	VAR robtarget OpenholeUD_5476 := [[469.92, -36.3, 185.04], [0.127117, 0.695587, 0.707021, -0.011034], [0,0,0,0], [9E9, 9E9, 9E9, 9E9, 9E9, 9E9]];
	VAR robtarget OpenholeUD_5477 := [[465.97, -36.3, 184.38], [0.114661, 0.697748, 0.707103, 0.002317], [0,0,0,0], [9E9, 9E9, 9E9, 9E9, 9E9, 9E9]];
	VAR robtarget OpenholeUD_5478 := [[462.03, -36.3, 183.73], [0.101936, 0.699721, 0.706932, 0.015742], [0,0,0,0], [9E9, 9E9, 9E9, 9E9, 9E9, 9E9]];
	VAR robtarget OpenholeUD_5479 := [[458.08, -36.3, 183.07], [0.088974, 0.701487, 0.706504, 0.029202], [0,0,0,0], [9E9, 9E9, 9E9, 9E9, 9E9, 9E9]];
	VAR robtarget OpenholeUD_5480 := [[454.14, -36.3, 182.42], [0.075811, 0.703031, 0.705819, 0.042651], [0,0,0,0], [9E9, 9E9, 9E9, 9E9, 9E9, 9E9]];
	VAR robtarget OpenholeUD_5481 := [[450.19, -36.3, 181.76], [0.062487, 0.70434, 0.704882, 0.056046], [0,0,0,0], [9E9, 9E9, 9E9, 9E9, 9E9, 9E9]];
	VAR robtarget OpenholeUD_5482 := [[446.24, -36.3, 181.11], [0.049045, 0.705404, 0.703698, 0.069344], [0,0,0,0], [9E9, 9E9, 9E9, 9E9, 9E9, 9E9]];
	VAR robtarget OpenholeUD_5483 := [[442.3, -36.3, 180.45], [0.035527, 0.706214, 0.702277, 0.082504], [0,0,0,0], [9E9, 9E9, 9E9, 9E9, 9E9, 9E9]];
	VAR robtarget OpenholeUD_5484 := [[438.35, -36.3, 179.79], [0.021978, 0.706765, 0.70063, 0.095485], [0,0,0,0], [9E9, 9E9, 9E9, 9E9, 9E9, 9E9]];
	VAR robtarget OpenholeUD_5485 := [[434.41, -36.3, 179.14], [0.008444, 0.707056, 0.698772, 0.10825], [0,0,0,0], [9E9, 9E9, 9E9, 9E9, 9E9, 9E9]];
	VAR robtarget OpenholeUD_5486 := [[430.46, -36.3, 178.48], [-0.005032, 0.707089, 0.696718, 0.120767], [0,0,0,0], [9E9, 9E9, 9E9, 9E9, 9E9, 9E9]];
	VAR robtarget OpenholeUD_5487 := [[426.52, -36.3, 177.83], [-0.018407, 0.706867, 0.694485, 0.133005], [0,0,0,0], [9E9, 9E9, 9E9, 9E9, 9E9, 9E9]];
	VAR robtarget OpenholeUD_5488 := [[422.57, -36.3, 177.17], [-0.03164, 0.706399, 0.692093, 0.144938], [0,0,0,0], [9E9, 9E9, 9E9, 9E9, 9E9, 9E9]];
	VAR robtarget OpenholeUD_5489 := [[418.62, -36.3, 176.52], [-0.044695, 0.705693, 0.68956, 0.156545], [0,0,0,0], [9E9, 9E9, 9E9, 9E9, 9E9, 9E9]];
	VAR robtarget OpenholeUD_5490 := [[414.68, -36.3, 175.86], [-0.057536, 0.704762, 0.686906, 0.167808], [0,0,0,0], [9E9, 9E9, 9E9, 9E9, 9E9, 9E9]];
	VAR robtarget OpenholeUD_5491 := [[410.73, -36.3, 175.2], [-0.070134, 0.70362, 0.68415, 0.178714], [0,0,0,0], [9E9, 9E9, 9E9, 9E9, 9E9, 9E9]];
	VAR robtarget OpenholeUD_5492 := [[406.79, -36.3, 174.55], [-0.082462, 0.702282, 0.68131, 0.189254], [0,0,0,0], [9E9, 9E9, 9E9, 9E9, 9E9, 9E9]];
	VAR robtarget OpenholeUD_5493 := [[402.84, -36.3, 173.89], [-0.094498, 0.700764, 0.678404, 0.199421], [0,0,0,0], [9E9, 9E9, 9E9, 9E9, 9E9, 9E9]];
	VAR robtarget OpenholeUD_5494 := [[398.89, -36.3, 173.24], [-0.106223, 0.699083, 0.675448, 0.209213], [0,0,0,0], [9E9, 9E9, 9E9, 9E9, 9E9, 9E9]];
	VAR robtarget OpenholeUD_5495 := [[394.95, -36.3, 172.58], [-0.117622, 0.697255, 0.672458, 0.218631], [0,0,0,0], [9E9, 9E9, 9E9, 9E9, 9E9, 9E9]];
	VAR robtarget OpenholeUD_5496 := [[389.32, -36.3, 171.65], [-0.13331, 0.694427, 0.66816, 0.231434], [0,0,0,0], [9E9, 9E9, 9E9, 9E9, 9E9, 9E9]];
	VAR robtarget OpenholeUD_5497 := [[385.32, -36.3, 171.66], [-0.183051, 0.683002, 0.683002, 0.183051], [0,0,0,0], [9E9, 9E9, 9E9, 9E9, 9E9, 9E9]];
	VAR robtarget OpenholeUD_5498 := [[381.32, -36.3, 171.67], [-0.183051, 0.683002, 0.683002, 0.183051], [0,0,0,0], [9E9, 9E9, 9E9, 9E9, 9E9, 9E9]];
	VAR robtarget OpenholeUD_5499 := [[377.32, -36.3, 171.68], [-0.183051, 0.683002, 0.683002, 0.183051], [0,0,0,0], [9E9, 9E9, 9E9, 9E9, 9E9, 9E9]];
	VAR robtarget OpenholeUD_5500 := [[373.32, -36.3, 171.7], [-0.183051, 0.683002, 0.683002, 0.183051], [0,0,0,0], [9E9, 9E9, 9E9, 9E9, 9E9, 9E9]];
	VAR robtarget OpenholeUD_5501 := [[369.32, -36.3, 171.71], [-0.183051, 0.683002, 0.683002, 0.183051], [0,0,0,0], [9E9, 9E9, 9E9, 9E9, 9E9, 9E9]];
	VAR robtarget OpenholeUD_5502 := [[369.32, -36.3, 171.71], [-0.183051, 0.683002, 0.683002, 0.183051], [0,0,0,0], [9E9, 9E9, 9E9, 9E9, 9E9, 9E9]];
	VAR robtarget OpenholeUD_5503 := [[369.31, -37.5, 171.02], [-0.183051, 0.683002, 0.683002, 0.183051], [0,0,0,0], [9E9, 9E9, 9E9, 9E9, 9E9, 9E9]];
	VAR robtarget OpenholeUD_5504 := [[373.31, -37.5, 171], [-0.183051, 0.683002, 0.683002, 0.183051], [0,0,0,0], [9E9, 9E9, 9E9, 9E9, 9E9, 9E9]];
	VAR robtarget OpenholeUD_5505 := [[377.31, -37.5, 170.99], [-0.183051, 0.683002, 0.683002, 0.183051], [0,0,0,0], [9E9, 9E9, 9E9, 9E9, 9E9, 9E9]];
	VAR robtarget OpenholeUD_5506 := [[381.31, -37.5, 170.98], [-0.183051, 0.683002, 0.683002, 0.183051], [0,0,0,0], [9E9, 9E9, 9E9, 9E9, 9E9, 9E9]];
	VAR robtarget OpenholeUD_5507 := [[385.31, -37.5, 170.97], [-0.183051, 0.683002, 0.683002, 0.183051], [0,0,0,0], [9E9, 9E9, 9E9, 9E9, 9E9, 9E9]];
	VAR robtarget OpenholeUD_5508 := [[389.31, -37.5, 170.95], [-0.129902, 0.695072, 0.667021, 0.234697], [0,0,0,0], [9E9, 9E9, 9E9, 9E9, 9E9, 9E9]];
	VAR robtarget OpenholeUD_5509 := [[393.25, -37.5, 171.65], [-0.118943, 0.697031, 0.670055, 0.225889], [0,0,0,0], [9E9, 9E9, 9E9, 9E9, 9E9, 9E9]];
	VAR robtarget OpenholeUD_5510 := [[397.19, -37.5, 172.35], [-0.107648, 0.698865, 0.673079, 0.216713], [0,0,0,0], [9E9, 9E9, 9E9, 9E9, 9E9, 9E9]];
	VAR robtarget OpenholeUD_5511 := [[401.13, -37.5, 173.05], [-0.096026, 0.700556, 0.676079, 0.207165], [0,0,0,0], [9E9, 9E9, 9E9, 9E9, 9E9, 9E9]];
	VAR robtarget OpenholeUD_5512 := [[405.07, -37.5, 173.75], [-0.084089, 0.702089, 0.679041, 0.197241], [0,0,0,0], [9E9, 9E9, 9E9, 9E9, 9E9, 9E9]];
	VAR robtarget OpenholeUD_5513 := [[409, -37.5, 174.45], [-0.071857, 0.703446, 0.681948, 0.186942], [0,0,0,0], [9E9, 9E9, 9E9, 9E9, 9E9, 9E9]];
	VAR robtarget OpenholeUD_5514 := [[412.94, -37.5, 175.15], [-0.059348, 0.704612, 0.684783, 0.176273], [0,0,0,0], [9E9, 9E9, 9E9, 9E9, 9E9, 9E9]];
	VAR robtarget OpenholeUD_5515 := [[416.88, -37.5, 175.85], [-0.04659, 0.70557, 0.687529, 0.165241], [0,0,0,0], [9E9, 9E9, 9E9, 9E9, 9E9, 9E9]];
	VAR robtarget OpenholeUD_5516 := [[420.82, -37.5, 176.55], [-0.03361, 0.706308, 0.690166, 0.153855], [0,0,0,0], [9E9, 9E9, 9E9, 9E9, 9E9, 9E9]];
	VAR robtarget OpenholeUD_5517 := [[424.76, -37.5, 177.25], [-0.020441, 0.706811, 0.692675, 0.142133], [0,0,0,0], [9E9, 9E9, 9E9, 9E9, 9E9, 9E9]];
	VAR robtarget OpenholeUD_5518 := [[428.7, -37.5, 177.95], [-0.00712, 0.707071, 0.695037, 0.130091], [0,0,0,0], [9E9, 9E9, 9E9, 9E9, 9E9, 9E9]];
	VAR robtarget OpenholeUD_5519 := [[432.63, -37.5, 178.65], [0.006313, 0.707079, 0.697233, 0.117755], [0,0,0,0], [9E9, 9E9, 9E9, 9E9, 9E9, 9E9]];
	VAR robtarget OpenholeUD_5520 := [[436.57, -37.5, 179.35], [0.019818, 0.706829, 0.699245, 0.105152], [0,0,0,0], [9E9, 9E9, 9E9, 9E9, 9E9, 9E9]];
	VAR robtarget OpenholeUD_5521 := [[440.51, -37.5, 180.05], [0.03335, 0.70632, 0.701055, 0.092312], [0,0,0,0], [9E9, 9E9, 9E9, 9E9, 9E9, 9E9]];
	VAR robtarget OpenholeUD_5522 := [[444.45, -37.5, 180.75], [0.046866, 0.705552, 0.702649, 0.079272], [0,0,0,0], [9E9, 9E9, 9E9, 9E9, 9E9, 9E9]];
	VAR robtarget OpenholeUD_5523 := [[448.39, -37.5, 181.45], [0.06032, 0.704529, 0.704013, 0.066068], [0,0,0,0], [9E9, 9E9, 9E9, 9E9, 9E9, 9E9]];
	VAR robtarget OpenholeUD_5524 := [[452.33, -37.5, 182.15], [0.073668, 0.703259, 0.705137, 0.052743], [0,0,0,0], [9E9, 9E9, 9E9, 9E9, 9E9, 9E9]];
	VAR robtarget OpenholeUD_5525 := [[456.26, -37.5, 182.85], [0.086868, 0.701751, 0.706012, 0.039337], [0,0,0,0], [9E9, 9E9, 9E9, 9E9, 9E9, 9E9]];
	VAR robtarget OpenholeUD_5526 := [[460.2, -37.5, 183.55], [0.09988, 0.700017, 0.706633, 0.025894], [0,0,0,0], [9E9, 9E9, 9E9, 9E9, 9E9, 9E9]];
	VAR robtarget OpenholeUD_5527 := [[464.14, -37.5, 184.25], [0.112666, 0.698073, 0.706997, 0.012458], [0,0,0,0], [9E9, 9E9, 9E9, 9E9, 9E9, 9E9]];
	VAR robtarget OpenholeUD_5528 := [[468.08, -37.5, 184.95], [0.125192, 0.695936, 0.707106, -0.000928], [0,0,0,0], [9E9, 9E9, 9E9, 9E9, 9E9, 9E9]];
	VAR robtarget OpenholeUD_5529 := [[472.02, -37.5, 185.65], [0.13743, 0.693623, 0.706964, -0.014223], [0,0,0,0], [9E9, 9E9, 9E9, 9E9, 9E9, 9E9]];
	VAR robtarget OpenholeUD_5530 := [[475.96, -37.5, 186.35], [0.149352, 0.691154, 0.706576, -0.027387], [0,0,0,0], [9E9, 9E9, 9E9, 9E9, 9E9, 9E9]];
	VAR robtarget OpenholeUD_5531 := [[479.89, -37.5, 187.05], [0.160938, 0.688548, 0.705953, -0.040383], [0,0,0,0], [9E9, 9E9, 9E9, 9E9, 9E9, 9E9]];
	VAR robtarget OpenholeUD_5532 := [[483.83, -37.5, 187.75], [0.172171, 0.685826, 0.705104, -0.053177], [0,0,0,0], [9E9, 9E9, 9E9, 9E9, 9E9, 9E9]];
	VAR robtarget OpenholeUD_5533 := [[487.77, -37.5, 188.45], [0.183038, 0.683006, 0.704044, -0.06574], [0,0,0,0], [9E9, 9E9, 9E9, 9E9, 9E9, 9E9]];
	VAR robtarget OpenholeUD_5534 := [[491.71, -37.5, 189.15], [0.193531, 0.680107, 0.702787, -0.078043], [0,0,0,0], [9E9, 9E9, 9E9, 9E9, 9E9, 9E9]];
	VAR robtarget OpenholeUD_5535 := [[495.65, -37.5, 189.85], [0.203644, 0.677148, 0.701347, -0.090066], [0,0,0,0], [9E9, 9E9, 9E9, 9E9, 9E9, 9E9]];
	VAR robtarget OpenholeUD_5536 := [[499.59, -37.5, 190.55], [0.213376, 0.674144, 0.699742, -0.101788], [0,0,0,0], [9E9, 9E9, 9E9, 9E9, 9E9, 9E9]];
	VAR robtarget OpenholeUD_5537 := [[503.52, -37.5, 191.25], [0.222729, 0.671112, 0.697988, -0.113195], [0,0,0,0], [9E9, 9E9, 9E9, 9E9, 9E9, 9E9]];
	VAR robtarget OpenholeUD_5538 := [[509.38, -37.5, 192.29], [0.183051, 0.683002, 0.683002, -0.183051], [0,0,0,0], [9E9, 9E9, 9E9, 9E9, 9E9, 9E9]];
	VAR robtarget OpenholeUD_5539 := [[513.38, -37.5, 192.28], [0.183051, 0.683002, 0.683002, -0.183051], [0,0,0,0], [9E9, 9E9, 9E9, 9E9, 9E9, 9E9]];
	VAR robtarget OpenholeUD_5540 := [[517.38, -37.5, 192.26], [0.183051, 0.683002, 0.683002, -0.183051], [0,0,0,0], [9E9, 9E9, 9E9, 9E9, 9E9, 9E9]];
	VAR robtarget OpenholeUD_5541 := [[521.38, -37.5, 192.25], [0.183051, 0.683002, 0.683002, -0.183051], [0,0,0,0], [9E9, 9E9, 9E9, 9E9, 9E9, 9E9]];
	VAR robtarget OpenholeUD_5542 := [[529.38, -37.5, 192.23], [0.183051, 0.683002, 0.683002, -0.183051], [0,0,0,0], [9E9, 9E9, 9E9, 9E9, 9E9, 9E9]];
	VAR robtarget OpenholeUD_5543 := [[529.38, -37.5, 192.23], [0.183051, 0.683002, 0.683002, -0.183051], [0,0,0,0], [9E9, 9E9, 9E9, 9E9, 9E9, 9E9]];
	VAR robtarget OpenholeUD_5544 := [[529.38, -38.7, 192.92], [0.183051, 0.683002, 0.683002, -0.183051], [0,0,0,0], [9E9, 9E9, 9E9, 9E9, 9E9, 9E9]];
	VAR robtarget OpenholeUD_5545 := [[525.38, -38.7, 192.93], [0.183051, 0.683002, 0.683002, -0.183051], [0,0,0,0], [9E9, 9E9, 9E9, 9E9, 9E9, 9E9]];
	VAR robtarget OpenholeUD_5546 := [[521.38, -38.7, 192.95], [0.183051, 0.683002, 0.683002, -0.183051], [0,0,0,0], [9E9, 9E9, 9E9, 9E9, 9E9, 9E9]];
	VAR robtarget OpenholeUD_5547 := [[517.38, -38.7, 192.96], [0.183051, 0.683002, 0.683002, -0.183051], [0,0,0,0], [9E9, 9E9, 9E9, 9E9, 9E9, 9E9]];
	VAR robtarget OpenholeUD_5548 := [[509.38, -38.7, 192.98], [0.183051, 0.683002, 0.683002, -0.183051], [0,0,0,0], [9E9, 9E9, 9E9, 9E9, 9E9, 9E9]];
	VAR robtarget OpenholeUD_5549 := [[505.45, -38.7, 192.24], [0.230297, 0.668553, 0.697618, -0.115451], [0,0,0,0], [9E9, 9E9, 9E9, 9E9, 9E9, 9E9]];
	VAR robtarget OpenholeUD_5550 := [[501.52, -38.7, 191.5], [0.221203, 0.671617, 0.699391, -0.104175], [0,0,0,0], [9E9, 9E9, 9E9, 9E9, 9E9, 9E9]];
	VAR robtarget OpenholeUD_5551 := [[497.59, -38.7, 190.75], [0.211734, 0.674662, 0.70102, -0.092579], [0,0,0,0], [9E9, 9E9, 9E9, 9E9, 9E9, 9E9]];
	VAR robtarget OpenholeUD_5552 := [[493.66, -38.7, 190.01], [0.201886, 0.677674, 0.702489, -0.080676], [0,0,0,0], [9E9, 9E9, 9E9, 9E9, 9E9, 9E9]];
	VAR robtarget OpenholeUD_5553 := [[489.73, -38.7, 189.26], [0.19166, 0.680637, 0.703783, -0.068482], [0,0,0,0], [9E9, 9E9, 9E9, 9E9, 9E9, 9E9]];
	VAR robtarget OpenholeUD_5554 := [[485.8, -38.7, 188.52], [0.181059, 0.683533, 0.704884, -0.056019], [0,0,0,0], [9E9, 9E9, 9E9, 9E9, 9E9, 9E9]];
	VAR robtarget OpenholeUD_5555 := [[481.87, -38.7, 187.78], [0.170089, 0.686345, 0.705779, -0.04331], [0,0,0,0], [9E9, 9E9, 9E9, 9E9, 9E9, 9E9]];
	VAR robtarget OpenholeUD_5556 := [[477.94, -38.7, 187.03], [0.158761, 0.689054, 0.706454, -0.030385], [0,0,0,0], [9E9, 9E9, 9E9, 9E9, 9E9, 9E9]];
	VAR robtarget OpenholeUD_5557 := [[474.01, -38.7, 186.29], [0.14709, 0.691639, 0.706896, -0.017277], [0,0,0,0], [9E9, 9E9, 9E9, 9E9, 9E9, 9E9]];
	VAR robtarget OpenholeUD_5558 := [[470.08, -38.7, 185.55], [0.135093, 0.694082, 0.707095, -0.004019], [0,0,0,0], [9E9, 9E9, 9E9, 9E9, 9E9, 9E9]];
	VAR robtarget OpenholeUD_5559 := [[466.15, -38.7, 184.8], [0.122794, 0.696363, 0.707045, 0.009348], [0,0,0,0], [9E9, 9E9, 9E9, 9E9, 9E9, 9E9]];
	VAR robtarget OpenholeUD_5560 := [[462.22, -38.7, 184.06], [0.110221, 0.698464, 0.70674, 0.022784], [0,0,0,0], [9E9, 9E9, 9E9, 9E9, 9E9, 9E9]];
	VAR robtarget OpenholeUD_5561 := [[458.29, -38.7, 183.31], [0.097404, 0.700366, 0.706177, 0.036247], [0,0,0,0], [9E9, 9E9, 9E9, 9E9, 9E9, 9E9]];
	VAR robtarget OpenholeUD_5562 := [[454.36, -38.7, 182.57], [0.084378, 0.702054, 0.705358, 0.049693], [0,0,0,0], [9E9, 9E9, 9E9, 9E9, 9E9, 9E9]];
	VAR robtarget OpenholeUD_5563 := [[450.43, -38.7, 181.83], [0.071182, 0.703515, 0.704288, 0.063078], [0,0,0,0], [9E9, 9E9, 9E9, 9E9, 9E9, 9E9]];
	VAR robtarget OpenholeUD_5564 := [[446.5, -38.7, 181.08], [0.057824, 0.704738, 0.702975, 0.076328], [0,0,0,0], [9E9, 9E9, 9E9, 9E9, 9E9, 9E9]];
	VAR robtarget OpenholeUD_5565 := [[442.57, -38.7, 180.34], [0.044363, 0.705714, 0.70143, 0.089417], [0,0,0,0], [9E9, 9E9, 9E9, 9E9, 9E9, 9E9]];
	VAR robtarget OpenholeUD_5566 := [[438.64, -38.7, 179.59], [0.030855, 0.706433, 0.699665, 0.102319], [0,0,0,0], [9E9, 9E9, 9E9, 9E9, 9E9, 9E9]];
	VAR robtarget OpenholeUD_5567 := [[434.71, -38.7, 178.85], [0.017344, 0.706894, 0.697693, 0.114998], [0,0,0,0], [9E9, 9E9, 9E9, 9E9, 9E9, 9E9]];
	VAR robtarget OpenholeUD_5568 := [[430.78, -38.7, 178.11], [0.003876, 0.707096, 0.695531, 0.127421], [0,0,0,0], [9E9, 9E9, 9E9, 9E9, 9E9, 9E9]];
	VAR robtarget OpenholeUD_5569 := [[426.85, -38.7, 177.36], [-0.009509, 0.707043, 0.693198, 0.139559], [0,0,0,0], [9E9, 9E9, 9E9, 9E9, 9E9, 9E9]];
	VAR robtarget OpenholeUD_5570 := [[422.92, -38.7, 176.62], [-0.022767, 0.70674, 0.690711, 0.151387], [0,0,0,0], [9E9, 9E9, 9E9, 9E9, 9E9, 9E9]];
	VAR robtarget OpenholeUD_5571 := [[418.99, -38.7, 175.88], [-0.035863, 0.706197, 0.688091, 0.162884], [0,0,0,0], [9E9, 9E9, 9E9, 9E9, 9E9, 9E9]];
	VAR robtarget OpenholeUD_5572 := [[415.06, -38.7, 175.13], [-0.048759, 0.705424, 0.685356, 0.174033], [0,0,0,0], [9E9, 9E9, 9E9, 9E9, 9E9, 9E9]];
	VAR robtarget OpenholeUD_5573 := [[411.13, -38.7, 174.39], [-0.061426, 0.704434, 0.682525, 0.184823], [0,0,0,0], [9E9, 9E9, 9E9, 9E9, 9E9, 9E9]];
	VAR robtarget OpenholeUD_5574 := [[407.2, -38.7, 173.64], [-0.073836, 0.703241, 0.679618, 0.195243], [0,0,0,0], [9E9, 9E9, 9E9, 9E9, 9E9, 9E9]];
	VAR robtarget OpenholeUD_5575 := [[403.27, -38.7, 172.9], [-0.085964, 0.701862, 0.676651, 0.20529], [0,0,0,0], [9E9, 9E9, 9E9, 9E9, 9E9, 9E9]];
	VAR robtarget OpenholeUD_5576 := [[399.34, -38.7, 172.16], [-0.097792, 0.700312, 0.673641, 0.214961], [0,0,0,0], [9E9, 9E9, 9E9, 9E9, 9E9, 9E9]];
	VAR robtarget OpenholeUD_5577 := [[395.41, -38.7, 171.41], [-0.109303, 0.698608, 0.670603, 0.224258], [0,0,0,0], [9E9, 9E9, 9E9, 9E9, 9E9, 9E9]];
	VAR robtarget OpenholeUD_5578 := [[389.31, -38.7, 170.26], [-0.126502, 0.695699, 0.66587, 0.237944], [0,0,0,0], [9E9, 9E9, 9E9, 9E9, 9E9, 9E9]];
	VAR robtarget OpenholeUD_5579 := [[385.31, -38.7, 170.27], [-0.183051, 0.683002, 0.683002, 0.183051], [0,0,0,0], [9E9, 9E9, 9E9, 9E9, 9E9, 9E9]];
	VAR robtarget OpenholeUD_5580 := [[381.31, -38.7, 170.29], [-0.183051, 0.683002, 0.683002, 0.183051], [0,0,0,0], [9E9, 9E9, 9E9, 9E9, 9E9, 9E9]];
	VAR robtarget OpenholeUD_5581 := [[377.31, -38.7, 170.3], [-0.183051, 0.683002, 0.683002, 0.183051], [0,0,0,0], [9E9, 9E9, 9E9, 9E9, 9E9, 9E9]];
	VAR robtarget OpenholeUD_5582 := [[373.31, -38.7, 170.31], [-0.183051, 0.683002, 0.683002, 0.183051], [0,0,0,0], [9E9, 9E9, 9E9, 9E9, 9E9, 9E9]];
	VAR robtarget OpenholeUD_5583 := [[369.31, -38.7, 170.32], [-0.183051, 0.683002, 0.683002, 0.183051], [0,0,0,0], [9E9, 9E9, 9E9, 9E9, 9E9, 9E9]];
	VAR robtarget OpenholeUD_5584 := [[369.31, -38.7, 170.32], [-0.183051, 0.683002, 0.683002, 0.183051], [0,0,0,0], [9E9, 9E9, 9E9, 9E9, 9E9, 9E9]];
	VAR robtarget OpenholeUD_5585 := [[369.31, -38.7, 170.44], [-0.183051, 0.683002, 0.683002, 0.183051], [0,0,0,0], [9E9, 9E9, 9E9, 9E9, 9E9, 9E9]];
	VAR robtarget OpenholeUD_5586 := [[373.31, -38.7, 170.43], [-0.183051, 0.683002, 0.683002, 0.183051], [0,0,0,0], [9E9, 9E9, 9E9, 9E9, 9E9, 9E9]];
	VAR robtarget OpenholeUD_5587 := [[377.31, -38.7, 170.42], [-0.183051, 0.683002, 0.683002, 0.183051], [0,0,0,0], [9E9, 9E9, 9E9, 9E9, 9E9, 9E9]];
	VAR robtarget OpenholeUD_5588 := [[381.31, -38.7, 170.41], [-0.183051, 0.683002, 0.683002, 0.183051], [0,0,0,0], [9E9, 9E9, 9E9, 9E9, 9E9, 9E9]];
	VAR robtarget OpenholeUD_5589 := [[385.31, -38.7, 170.39], [-0.183051, 0.683002, 0.683002, 0.183051], [0,0,0,0], [9E9, 9E9, 9E9, 9E9, 9E9, 9E9]];
	VAR robtarget OpenholeUD_5590 := [[389.31, -38.7, 170.38], [-0.126598, 0.695682, 0.665932, 0.237771], [0,0,0,0], [9E9, 9E9, 9E9, 9E9, 9E9, 9E9]];
	VAR robtarget OpenholeUD_5591 := [[393.24, -38.7, 171.12], [-0.115595, 0.697594, 0.668983, 0.229046], [0,0,0,0], [9E9, 9E9, 9E9, 9E9, 9E9, 9E9]];
	VAR robtarget OpenholeUD_5592 := [[397.17, -38.7, 171.87], [-0.104257, 0.699379, 0.672027, 0.219954], [0,0,0,0], [9E9, 9E9, 9E9, 9E9, 9E9, 9E9]];
	VAR robtarget OpenholeUD_5593 := [[401.1, -38.7, 172.61], [-0.092594, 0.701018, 0.675051, 0.210491], [0,0,0,0], [9E9, 9E9, 9E9, 9E9, 9E9, 9E9]];
	VAR robtarget OpenholeUD_5594 := [[405.03, -38.7, 173.36], [-0.08062, 0.702496, 0.67804, 0.200653], [0,0,0,0], [9E9, 9E9, 9E9, 9E9, 9E9, 9E9]];
	VAR robtarget OpenholeUD_5595 := [[408.96, -38.7, 174.1], [-0.068353, 0.703795, 0.680979, 0.190441], [0,0,0,0], [9E9, 9E9, 9E9, 9E9, 9E9, 9E9]];
	VAR robtarget OpenholeUD_5596 := [[412.89, -38.7, 174.84], [-0.055814, 0.704901, 0.68385, 0.179857], [0,0,0,0], [9E9, 9E9, 9E9, 9E9, 9E9, 9E9]];
	VAR robtarget OpenholeUD_5597 := [[416.82, -38.7, 175.59], [-0.043029, 0.705796, 0.686636, 0.16891], [0,0,0,0], [9E9, 9E9, 9E9, 9E9, 9E9, 9E9]];
	VAR robtarget OpenholeUD_5598 := [[420.75, -38.7, 176.33], [-0.030027, 0.706469, 0.689318, 0.157609], [0,0,0,0], [9E9, 9E9, 9E9, 9E9, 9E9, 9E9]];
	VAR robtarget OpenholeUD_5599 := [[424.68, -38.7, 177.07], [-0.01684, 0.706906, 0.691877, 0.145968], [0,0,0,0], [9E9, 9E9, 9E9, 9E9, 9E9, 9E9]];
	VAR robtarget OpenholeUD_5600 := [[428.61, -38.7, 177.82], [-0.003507, 0.707098, 0.694293, 0.134007], [0,0,0,0], [9E9, 9E9, 9E9, 9E9, 9E9, 9E9]];
	VAR robtarget OpenholeUD_5601 := [[432.54, -38.7, 178.56], [0.009934, 0.707037, 0.696547, 0.121747], [0,0,0,0], [9E9, 9E9, 9E9, 9E9, 9E9, 9E9]];
	VAR robtarget OpenholeUD_5602 := [[436.47, -38.7, 179.31], [0.023442, 0.706718, 0.698621, 0.109216], [0,0,0,0], [9E9, 9E9, 9E9, 9E9, 9E9, 9E9]];
	VAR robtarget OpenholeUD_5603 := [[440.4, -38.7, 180.05], [0.036971, 0.70614, 0.700499, 0.096444], [0,0,0,0], [9E9, 9E9, 9E9, 9E9, 9E9, 9E9]];
	VAR robtarget OpenholeUD_5604 := [[444.33, -38.7, 180.79], [0.050478, 0.705303, 0.702163, 0.083465], [0,0,0,0], [9E9, 9E9, 9E9, 9E9, 9E9, 9E9]];
	VAR robtarget OpenholeUD_5605 := [[448.27, -38.7, 181.54], [0.063918, 0.704212, 0.703602, 0.070318], [0,0,0,0], [9E9, 9E9, 9E9, 9E9, 9E9, 9E9]];
	VAR robtarget OpenholeUD_5606 := [[452.2, -38.7, 182.28], [0.077204, 0.702879, 0.704806, 0.056999], [0,0,0,0], [9E9, 9E9, 9E9, 9E9, 9E9, 9E9]];
	VAR robtarget OpenholeUD_5607 := [[456.13, -38.7, 183.02], [0.090328, 0.701314, 0.705763, 0.043581], [0,0,0,0], [9E9, 9E9, 9E9, 9E9, 9E9, 9E9]];
	VAR robtarget OpenholeUD_5608 := [[460.06, -38.7, 183.77], [0.103263, 0.699526, 0.706465, 0.030122], [0,0,0,0], [9E9, 9E9, 9E9, 9E9, 9E9, 9E9]];
	VAR robtarget OpenholeUD_5609 := [[463.99, -38.7, 184.51], [0.115973, 0.697531, 0.70691, 0.016665], [0,0,0,0], [9E9, 9E9, 9E9, 9E9, 9E9, 9E9]];
	VAR robtarget OpenholeUD_5610 := [[467.92, -38.7, 185.26], [0.128426, 0.695347, 0.707099, 0.003255], [0,0,0,0], [9E9, 9E9, 9E9, 9E9, 9E9, 9E9]];
	VAR robtarget OpenholeUD_5611 := [[471.85, -38.7, 186], [0.14059, 0.69299, 0.707035, -0.010067], [0,0,0,0], [9E9, 9E9, 9E9, 9E9, 9E9, 9E9]];
	VAR robtarget OpenholeUD_5612 := [[475.78, -38.7, 186.74], [0.152441, 0.690479, 0.706724, -0.023262], [0,0,0,0], [9E9, 9E9, 9E9, 9E9, 9E9, 9E9]];
	VAR robtarget OpenholeUD_5613 := [[479.71, -38.7, 187.49], [0.163959, 0.687835, 0.706175, -0.036291], [0,0,0,0], [9E9, 9E9, 9E9, 9E9, 9E9, 9E9]];
	VAR robtarget OpenholeUD_5614 := [[483.64, -38.7, 188.23], [0.175126, 0.685077, 0.705399, -0.049121], [0,0,0,0], [9E9, 9E9, 9E9, 9E9, 9E9, 9E9]];
	VAR robtarget OpenholeUD_5615 := [[487.57, -38.7, 188.97], [0.185929, 0.682225, 0.704408, -0.061721], [0,0,0,0], [9E9, 9E9, 9E9, 9E9, 9E9, 9E9]];
	VAR robtarget OpenholeUD_5616 := [[491.5, -38.7, 189.72], [0.19636, 0.679296, 0.703217, -0.074065], [0,0,0,0], [9E9, 9E9, 9E9, 9E9, 9E9, 9E9]];
	VAR robtarget OpenholeUD_5617 := [[495.43, -38.7, 190.46], [0.206414, 0.676309, 0.701842, -0.086129], [0,0,0,0], [9E9, 9E9, 9E9, 9E9, 9E9, 9E9]];
	VAR robtarget OpenholeUD_5618 := [[499.36, -38.7, 191.21], [0.216089, 0.67328, 0.700298, -0.097894], [0,0,0,0], [9E9, 9E9, 9E9, 9E9, 9E9, 9E9]];
	VAR robtarget OpenholeUD_5619 := [[503.29, -38.7, 191.95], [0.225387, 0.670224, 0.698601, -0.109346], [0,0,0,0], [9E9, 9E9, 9E9, 9E9, 9E9, 9E9]];
	VAR robtarget OpenholeUD_5620 := [[509.38, -38.7, 193.1], [0.183051, 0.683002, 0.683002, -0.183051], [0,0,0,0], [9E9, 9E9, 9E9, 9E9, 9E9, 9E9]];
	VAR robtarget OpenholeUD_5621 := [[513.38, -38.7, 193.09], [0.183051, 0.683002, 0.683002, -0.183051], [0,0,0,0], [9E9, 9E9, 9E9, 9E9, 9E9, 9E9]];
	VAR robtarget OpenholeUD_5622 := [[517.38, -38.7, 193.08], [0.183051, 0.683002, 0.683002, -0.183051], [0,0,0,0], [9E9, 9E9, 9E9, 9E9, 9E9, 9E9]];
	VAR robtarget OpenholeUD_5623 := [[521.38, -38.7, 193.07], [0.183051, 0.683002, 0.683002, -0.183051], [0,0,0,0], [9E9, 9E9, 9E9, 9E9, 9E9, 9E9]];
	VAR robtarget OpenholeUD_5624 := [[525.38, -38.7, 193.05], [0.183051, 0.683002, 0.683002, -0.183051], [0,0,0,0], [9E9, 9E9, 9E9, 9E9, 9E9, 9E9]];
	VAR robtarget OpenholeUD_5625 := [[529.38, -38.7, 193.04], [0.183051, 0.683002, 0.683002, -0.183051], [0,0,0,0], [9E9, 9E9, 9E9, 9E9, 9E9, 9E9]];
	VAR robtarget OpenholeUD_5626 := [[529.38, -38.7, 193.04], [0.183051, 0.683002, 0.683002, -0.183051], [0,0,0,0], [9E9, 9E9, 9E9, 9E9, 9E9, 9E9]];
	VAR robtarget OpenholeUD_5627 := [[529.38, -37.5, 192.35], [0.183051, 0.683002, 0.683002, -0.183051], [0,0,0,0], [9E9, 9E9, 9E9, 9E9, 9E9, 9E9]];
	VAR robtarget OpenholeUD_5628 := [[525.38, -37.5, 192.36], [0.183051, 0.683002, 0.683002, -0.183051], [0,0,0,0], [9E9, 9E9, 9E9, 9E9, 9E9, 9E9]];
	VAR robtarget OpenholeUD_5629 := [[521.38, -37.5, 192.37], [0.183051, 0.683002, 0.683002, -0.183051], [0,0,0,0], [9E9, 9E9, 9E9, 9E9, 9E9, 9E9]];
	VAR robtarget OpenholeUD_5630 := [[517.38, -37.5, 192.38], [0.183051, 0.683002, 0.683002, -0.183051], [0,0,0,0], [9E9, 9E9, 9E9, 9E9, 9E9, 9E9]];
	VAR robtarget OpenholeUD_5631 := [[513.38, -37.5, 192.4], [0.183051, 0.683002, 0.683002, -0.183051], [0,0,0,0], [9E9, 9E9, 9E9, 9E9, 9E9, 9E9]];
	VAR robtarget OpenholeUD_5632 := [[509.38, -37.5, 192.41], [0.183051, 0.683002, 0.683002, -0.183051], [0,0,0,0], [9E9, 9E9, 9E9, 9E9, 9E9, 9E9]];
	VAR robtarget OpenholeUD_5633 := [[505.44, -37.5, 191.71], [0.227323, 0.66957, 0.6971, -0.118541], [0,0,0,0], [9E9, 9E9, 9E9, 9E9, 9E9, 9E9]];
	VAR robtarget OpenholeUD_5634 := [[501.5, -37.5, 191.01], [0.218153, 0.672614, 0.698918, -0.107299], [0,0,0,0], [9E9, 9E9, 9E9, 9E9, 9E9, 9E9]];
	VAR robtarget OpenholeUD_5635 := [[497.57, -37.5, 190.31], [0.208605, 0.675636, 0.700596, -0.095736], [0,0,0,0], [9E9, 9E9, 9E9, 9E9, 9E9, 9E9]];
	VAR robtarget OpenholeUD_5636 := [[493.63, -37.5, 189.61], [0.198676, 0.678622, 0.702116, -0.083866], [0,0,0,0], [9E9, 9E9, 9E9, 9E9, 9E9, 9E9]];
	VAR robtarget OpenholeUD_5637 := [[489.69, -37.5, 188.91], [0.188365, 0.681556, 0.703462, -0.071706], [0,0,0,0], [9E9, 9E9, 9E9, 9E9, 9E9, 9E9]];
	VAR robtarget OpenholeUD_5638 := [[485.75, -37.5, 188.21], [0.177675, 0.684421, 0.704618, -0.059276], [0,0,0,0], [9E9, 9E9, 9E9, 9E9, 9E9, 9E9]];
	VAR robtarget OpenholeUD_5639 := [[481.81, -37.5, 187.51], [0.166614, 0.687197, 0.705569, -0.046603], [0,0,0,0], [9E9, 9E9, 9E9, 9E9, 9E9, 9E9]];
	VAR robtarget OpenholeUD_5640 := [[477.87, -37.5, 186.81], [0.155191, 0.689866, 0.706303, -0.033713], [0,0,0,0], [9E9, 9E9, 9E9, 9E9, 9E9, 9E9]];
	VAR robtarget OpenholeUD_5641 := [[473.94, -37.5, 186.11], [0.143423, 0.692409, 0.706806, -0.020639], [0,0,0,0], [9E9, 9E9, 9E9, 9E9, 9E9, 9E9]];
	VAR robtarget OpenholeUD_5642 := [[470, -37.5, 185.41], [0.131328, 0.694804, 0.707068, -0.007417], [0,0,0,0], [9E9, 9E9, 9E9, 9E9, 9E9, 9E9]];
	VAR robtarget OpenholeUD_5643 := [[466.06, -37.5, 184.71], [0.118929, 0.697034, 0.707082, 0.005916], [0,0,0,0], [9E9, 9E9, 9E9, 9E9, 9E9, 9E9]];
	VAR robtarget OpenholeUD_5644 := [[462.12, -37.5, 184.01], [0.106254, 0.699078, 0.706843, 0.019319], [0,0,0,0], [9E9, 9E9, 9E9, 9E9, 9E9, 9E9]];
	VAR robtarget OpenholeUD_5645 := [[458.18, -37.5, 183.31], [0.093336, 0.70092, 0.706348, 0.032749], [0,0,0,0], [9E9, 9E9, 9E9, 9E9, 9E9, 9E9]];
	VAR robtarget OpenholeUD_5646 := [[454.25, -37.5, 182.61], [0.08021, 0.702543, 0.705598, 0.046164], [0,0,0,0], [9E9, 9E9, 9E9, 9E9, 9E9, 9E9]];
	VAR robtarget OpenholeUD_5647 := [[450.31, -37.5, 181.91], [0.066915, 0.703933, 0.704597, 0.05952], [0,0,0,0], [9E9, 9E9, 9E9, 9E9, 9E9, 9E9]];
	VAR robtarget OpenholeUD_5648 := [[446.37, -37.5, 181.21], [0.053494, 0.70508, 0.703352, 0.072775], [0,0,0,0], [9E9, 9E9, 9E9, 9E9, 9E9, 9E9]];
	VAR robtarget OpenholeUD_5649 := [[442.43, -37.5, 180.51], [0.039988, 0.705975, 0.701871, 0.085887], [0,0,0,0], [9E9, 9E9, 9E9, 9E9, 9E9, 9E9]];
	VAR robtarget OpenholeUD_5650 := [[438.49, -37.5, 179.81], [0.026444, 0.706612, 0.700168, 0.098817], [0,0,0,0], [9E9, 9E9, 9E9, 9E9, 9E9, 9E9]];
	VAR robtarget OpenholeUD_5651 := [[434.55, -37.5, 179.11], [0.012906, 0.706989, 0.698256, 0.111528], [0,0,0,0], [9E9, 9E9, 9E9, 9E9, 9E9, 9E9]];
	VAR robtarget OpenholeUD_5652 := [[430.62, -37.5, 178.41], [-0.000582, 0.707107, 0.696152, 0.123988], [0,0,0,0], [9E9, 9E9, 9E9, 9E9, 9E9, 9E9]];
	VAR robtarget OpenholeUD_5653 := [[426.68, -37.5, 177.71], [-0.013977, 0.706969, 0.693872, 0.136166], [0,0,0,0], [9E9, 9E9, 9E9, 9E9, 9E9, 9E9]];
	VAR robtarget OpenholeUD_5654 := [[422.74, -37.5, 177.01], [-0.027238, 0.706582, 0.691437, 0.148039], [0,0,0,0], [9E9, 9E9, 9E9, 9E9, 9E9, 9E9]];
	VAR robtarget OpenholeUD_5655 := [[418.8, -37.5, 176.31], [-0.040327, 0.705956, 0.688864, 0.159584], [0,0,0,0], [9E9, 9E9, 9E9, 9E9, 9E9, 9E9]];
	VAR robtarget OpenholeUD_5656 := [[414.86, -37.5, 175.61], [-0.053209, 0.705102, 0.686173, 0.170784], [0,0,0,0], [9E9, 9E9, 9E9, 9E9, 9E9, 9E9]];
	VAR robtarget OpenholeUD_5657 := [[410.92, -37.5, 174.91], [-0.065854, 0.704034, 0.683383, 0.181626], [0,0,0,0], [9E9, 9E9, 9E9, 9E9, 9E9, 9E9]];
	VAR robtarget OpenholeUD_5658 := [[406.99, -37.5, 174.21], [-0.078233, 0.702766, 0.680512, 0.192102], [0,0,0,0], [9E9, 9E9, 9E9, 9E9, 9E9, 9E9]];
	VAR robtarget OpenholeUD_5659 := [[403.05, -37.5, 173.51], [-0.090326, 0.701314, 0.677578, 0.202206], [0,0,0,0], [9E9, 9E9, 9E9, 9E9, 9E9, 9E9]];
	VAR robtarget OpenholeUD_5660 := [[399.11, -37.5, 172.81], [-0.102111, 0.699695, 0.674598, 0.211936], [0,0,0,0], [9E9, 9E9, 9E9, 9E9, 9E9, 9E9]];
	VAR robtarget OpenholeUD_5661 := [[395.17, -37.5, 172.11], [-0.113574, 0.697926, 0.671587, 0.221292], [0,0,0,0], [9E9, 9E9, 9E9, 9E9, 9E9, 9E9]];
	VAR robtarget OpenholeUD_5662 := [[389.31, -37.5, 171.07], [-0.130002, 0.695054, 0.667082, 0.234524], [0,0,0,0], [9E9, 9E9, 9E9, 9E9, 9E9, 9E9]];
	VAR robtarget OpenholeUD_5663 := [[385.31, -37.5, 171.09], [-0.183051, 0.683002, 0.683002, 0.183051], [0,0,0,0], [9E9, 9E9, 9E9, 9E9, 9E9, 9E9]];
	VAR robtarget OpenholeUD_5664 := [[381.31, -37.5, 171.1], [-0.183051, 0.683002, 0.683002, 0.183051], [0,0,0,0], [9E9, 9E9, 9E9, 9E9, 9E9, 9E9]];
	VAR robtarget OpenholeUD_5665 := [[377.31, -37.5, 171.11], [-0.183051, 0.683002, 0.683002, 0.183051], [0,0,0,0], [9E9, 9E9, 9E9, 9E9, 9E9, 9E9]];
	VAR robtarget OpenholeUD_5666 := [[373.31, -37.5, 171.12], [-0.183051, 0.683002, 0.683002, 0.183051], [0,0,0,0], [9E9, 9E9, 9E9, 9E9, 9E9, 9E9]];
	VAR robtarget OpenholeUD_5667 := [[369.31, -37.5, 171.14], [-0.183051, 0.683002, 0.683002, 0.183051], [0,0,0,0], [9E9, 9E9, 9E9, 9E9, 9E9, 9E9]];
	VAR robtarget OpenholeUD_5668 := [[369.31, -37.5, 171.14], [-0.183051, 0.683002, 0.683002, 0.183051], [0,0,0,0], [9E9, 9E9, 9E9, 9E9, 9E9, 9E9]];
	VAR robtarget OpenholeUD_5669 := [[369.32, -36.3, 171.83], [-0.183051, 0.683002, 0.683002, 0.183051], [0,0,0,0], [9E9, 9E9, 9E9, 9E9, 9E9, 9E9]];
	VAR robtarget OpenholeUD_5670 := [[373.32, -36.3, 171.82], [-0.183051, 0.683002, 0.683002, 0.183051], [0,0,0,0], [9E9, 9E9, 9E9, 9E9, 9E9, 9E9]];
	VAR robtarget OpenholeUD_5671 := [[377.32, -36.3, 171.8], [-0.183051, 0.683002, 0.683002, 0.183051], [0,0,0,0], [9E9, 9E9, 9E9, 9E9, 9E9, 9E9]];
	VAR robtarget OpenholeUD_5672 := [[381.32, -36.3, 171.79], [-0.183051, 0.683002, 0.683002, 0.183051], [0,0,0,0], [9E9, 9E9, 9E9, 9E9, 9E9, 9E9]];
	VAR robtarget OpenholeUD_5673 := [[385.32, -36.3, 171.78], [-0.183051, 0.683002, 0.683002, 0.183051], [0,0,0,0], [9E9, 9E9, 9E9, 9E9, 9E9, 9E9]];
	VAR robtarget OpenholeUD_5674 := [[389.32, -36.3, 171.77], [-0.133413, 0.694407, 0.66822, 0.231262], [0,0,0,0], [9E9, 9E9, 9E9, 9E9, 9E9, 9E9]];
	VAR robtarget OpenholeUD_5675 := [[393.26, -36.3, 172.42], [-0.122491, 0.696417, 0.671231, 0.222372], [0,0,0,0], [9E9, 9E9, 9E9, 9E9, 9E9, 9E9]];
	VAR robtarget OpenholeUD_5676 := [[397.21, -36.3, 173.08], [-0.111228, 0.698304, 0.674228, 0.213113], [0,0,0,0], [9E9, 9E9, 9E9, 9E9, 9E9, 9E9]];
	VAR robtarget OpenholeUD_5677 := [[401.15, -36.3, 173.73], [-0.099633, 0.700052, 0.677196, 0.203482], [0,0,0,0], [9E9, 9E9, 9E9, 9E9, 9E9, 9E9]];
	VAR robtarget OpenholeUD_5678 := [[405.1, -36.3, 174.39], [-0.08772, 0.701645, 0.680122, 0.193477], [0,0,0,0], [9E9, 9E9, 9E9, 9E9, 9E9, 9E9]];
	VAR robtarget OpenholeUD_5679 := [[409.05, -36.3, 175.04], [-0.075505, 0.703064, 0.682989, 0.1831], [0,0,0,0], [9E9, 9E9, 9E9, 9E9, 9E9, 9E9]];
	VAR robtarget OpenholeUD_5680 := [[412.99, -36.3, 175.7], [-0.063009, 0.704294, 0.68578, 0.172354], [0,0,0,0], [9E9, 9E9, 9E9, 9E9, 9E9, 9E9]];
	VAR robtarget OpenholeUD_5681 := [[416.94, -36.3, 176.36], [-0.050257, 0.705319, 0.688476, 0.161248], [0,0,0,0], [9E9, 9E9, 9E9, 9E9, 9E9, 9E9]];
	VAR robtarget OpenholeUD_5682 := [[420.88, -36.3, 177.01], [-0.037277, 0.706124, 0.691059, 0.149793], [0,0,0,0], [9E9, 9E9, 9E9, 9E9, 9E9, 9E9]];
	VAR robtarget OpenholeUD_5683 := [[424.83, -36.3, 177.67], [-0.024102, 0.706696, 0.693509, 0.138005], [0,0,0,0], [9E9, 9E9, 9E9, 9E9, 9E9, 9E9]];
	VAR robtarget OpenholeUD_5684 := [[428.77, -36.3, 178.32], [-0.01077, 0.707025, 0.695808, 0.125903], [0,0,0,0], [9E9, 9E9, 9E9, 9E9, 9E9, 9E9]];
	VAR robtarget OpenholeUD_5685 := [[432.72, -36.3, 178.98], [0.002682, 0.707102, 0.697936, 0.113512], [0,0,0,0], [9E9, 9E9, 9E9, 9E9, 9E9, 9E9]];
	VAR robtarget OpenholeUD_5686 := [[436.67, -36.3, 179.63], [0.016212, 0.706921, 0.699877, 0.10086], [0,0,0,0], [9E9, 9E9, 9E9, 9E9, 9E9, 9E9]];
	VAR robtarget OpenholeUD_5687 := [[440.61, -36.3, 180.29], [0.029774, 0.70648, 0.701612, 0.087979], [0,0,0,0], [9E9, 9E9, 9E9, 9E9, 9E9, 9E9]];
	VAR robtarget OpenholeUD_5688 := [[444.56, -36.3, 180.95], [0.043325, 0.705778, 0.703128, 0.074904], [0,0,0,0], [9E9, 9E9, 9E9, 9E9, 9E9, 9E9]];
	VAR robtarget OpenholeUD_5689 := [[448.5, -36.3, 181.6], [0.05682, 0.70482, 0.704412, 0.061673], [0,0,0,0], [9E9, 9E9, 9E9, 9E9, 9E9, 9E9]];
	VAR robtarget OpenholeUD_5690 := [[452.45, -36.3, 182.26], [0.070214, 0.703612, 0.705453, 0.048328], [0,0,0,0], [9E9, 9E9, 9E9, 9E9, 9E9, 9E9]];
	VAR robtarget OpenholeUD_5691 := [[456.4, -36.3, 182.91], [0.083463, 0.702164, 0.706244, 0.034911], [0,0,0,0], [9E9, 9E9, 9E9, 9E9, 9E9, 9E9]];
	VAR robtarget OpenholeUD_5692 := [[460.34, -36.3, 183.57], [0.096528, 0.700487, 0.706781, 0.021466], [0,0,0,0], [9E9, 9E9, 9E9, 9E9, 9E9, 9E9]];
	VAR robtarget OpenholeUD_5693 := [[464.29, -36.3, 184.22], [0.109371, 0.698597, 0.707061, 0.008035], [0,0,0,0], [9E9, 9E9, 9E9, 9E9, 9E9, 9E9]];
	VAR robtarget OpenholeUD_5694 := [[468.23, -36.3, 184.88], [0.121956, 0.69651, 0.707087, -0.005339], [0,0,0,0], [9E9, 9E9, 9E9, 9E9, 9E9, 9E9]];
	VAR robtarget OpenholeUD_5695 := [[472.18, -36.3, 185.54], [0.134255, 0.694245, 0.706862, -0.018614], [0,0,0,0], [9E9, 9E9, 9E9, 9E9, 9E9, 9E9]];
	VAR robtarget OpenholeUD_5696 := [[476.13, -36.3, 186.19], [0.14624, 0.691819, 0.706394, -0.03175], [0,0,0,0], [9E9, 9E9, 9E9, 9E9, 9E9, 9E9]];
	VAR robtarget OpenholeUD_5697 := [[480.07, -36.3, 186.85], [0.157889, 0.689254, 0.705692, -0.044712], [0,0,0,0], [9E9, 9E9, 9E9, 9E9, 9E9, 9E9]];
	VAR robtarget OpenholeUD_5698 := [[484.02, -36.3, 187.5], [0.169187, 0.686568, 0.704768, -0.057467], [0,0,0,0], [9E9, 9E9, 9E9, 9E9, 9E9, 9E9]];
	VAR robtarget OpenholeUD_5699 := [[487.96, -36.3, 188.16], [0.180118, 0.683782, 0.703635, -0.069983], [0,0,0,0], [9E9, 9E9, 9E9, 9E9, 9E9, 9E9]];
	VAR robtarget OpenholeUD_5700 := [[491.91, -36.3, 188.81], [0.190676, 0.680913, 0.702308, -0.082237], [0,0,0,0], [9E9, 9E9, 9E9, 9E9, 9E9, 9E9]];
	VAR robtarget OpenholeUD_5701 := [[495.86, -36.3, 189.47], [0.200853, 0.677981, 0.700804, -0.094204], [0,0,0,0], [9E9, 9E9, 9E9, 9E9, 9E9, 9E9]];
	VAR robtarget OpenholeUD_5702 := [[499.8, -36.3, 190.13], [0.210649, 0.675002, 0.699137, -0.105868], [0,0,0,0], [9E9, 9E9, 9E9, 9E9, 9E9, 9E9]];
	VAR robtarget OpenholeUD_5703 := [[503.75, -36.3, 190.78], [0.220064, 0.671991, 0.697324, -0.117213], [0,0,0,0], [9E9, 9E9, 9E9, 9E9, 9E9, 9E9]];
	VAR robtarget OpenholeUD_5704 := [[509.38, -36.3, 191.72], [0.183051, 0.683002, 0.683002, -0.183051], [0,0,0,0], [9E9, 9E9, 9E9, 9E9, 9E9, 9E9]];
	VAR robtarget OpenholeUD_5705 := [[513.38, -36.3, 191.7], [0.183051, 0.683002, 0.683002, -0.183051], [0,0,0,0], [9E9, 9E9, 9E9, 9E9, 9E9, 9E9]];
	VAR robtarget OpenholeUD_5706 := [[517.38, -36.3, 191.69], [0.183051, 0.683002, 0.683002, -0.183051], [0,0,0,0], [9E9, 9E9, 9E9, 9E9, 9E9, 9E9]];
	VAR robtarget OpenholeUD_5707 := [[521.38, -36.3, 191.68], [0.183051, 0.683002, 0.683002, -0.183051], [0,0,0,0], [9E9, 9E9, 9E9, 9E9, 9E9, 9E9]];
	VAR robtarget OpenholeUD_5708 := [[525.38, -36.3, 191.67], [0.183051, 0.683002, 0.683002, -0.183051], [0,0,0,0], [9E9, 9E9, 9E9, 9E9, 9E9, 9E9]];
	VAR robtarget OpenholeUD_5709 := [[529.38, -36.3, 191.65], [0.183051, 0.683002, 0.683002, -0.183051], [0,0,0,0], [9E9, 9E9, 9E9, 9E9, 9E9, 9E9]];
	VAR robtarget OpenholeUD_5710 := [[529.38, -36.3, 191.65], [0.183051, 0.683002, 0.683002, -0.183051], [0,0,0,0], [9E9, 9E9, 9E9, 9E9, 9E9, 9E9]];
	VAR robtarget OpenholeUD_5711 := [[529.38, -35.1, 190.96], [0.183051, 0.683002, 0.683002, -0.183051], [0,0,0,0], [9E9, 9E9, 9E9, 9E9, 9E9, 9E9]];
	VAR robtarget OpenholeUD_5712 := [[525.38, -35.1, 190.97], [0.183051, 0.683002, 0.683002, -0.183051], [0,0,0,0], [9E9, 9E9, 9E9, 9E9, 9E9, 9E9]];
	VAR robtarget OpenholeUD_5713 := [[521.38, -35.1, 190.99], [0.183051, 0.683002, 0.683002, -0.183051], [0,0,0,0], [9E9, 9E9, 9E9, 9E9, 9E9, 9E9]];
	VAR robtarget OpenholeUD_5714 := [[517.38, -35.1, 191], [0.183051, 0.683002, 0.683002, -0.183051], [0,0,0,0], [9E9, 9E9, 9E9, 9E9, 9E9, 9E9]];
	VAR robtarget OpenholeUD_5715 := [[513.38, -35.1, 191.01], [0.183051, 0.683002, 0.683002, -0.183051], [0,0,0,0], [9E9, 9E9, 9E9, 9E9, 9E9, 9E9]];
	VAR robtarget OpenholeUD_5716 := [[509.38, -35.1, 191.02], [0.183051, 0.683002, 0.683002, -0.183051], [0,0,0,0], [9E9, 9E9, 9E9, 9E9, 9E9, 9E9]];
	VAR robtarget OpenholeUD_5717 := [[505.42, -35.1, 190.41], [0.220609, 0.671812, 0.6959, -0.12539], [0,0,0,0], [9E9, 9E9, 9E9, 9E9, 9E9, 9E9]];
	VAR robtarget OpenholeUD_5718 := [[501.47, -35.1, 189.8], [0.211271, 0.674807, 0.69782, -0.114225], [0,0,0,0], [9E9, 9E9, 9E9, 9E9, 9E9, 9E9]];
	VAR robtarget OpenholeUD_5719 := [[497.52, -35.1, 189.19], [0.201553, 0.677773, 0.699604, -0.102732], [0,0,0,0], [9E9, 9E9, 9E9, 9E9, 9E9, 9E9]];
	VAR robtarget OpenholeUD_5720 := [[493.56, -35.1, 188.58], [0.191455, 0.680694, 0.701236, -0.090926], [0,0,0,0], [9E9, 9E9, 9E9, 9E9, 9E9, 9E9]];
	VAR robtarget OpenholeUD_5721 := [[489.61, -35.1, 187.97], [0.180977, 0.683555, 0.7027, -0.078821], [0,0,0,0], [9E9, 9E9, 9E9, 9E9, 9E9, 9E9]];
	VAR robtarget OpenholeUD_5722 := [[485.66, -35.1, 187.36], [0.170122, 0.686337, 0.703979, -0.066439], [0,0,0,0], [9E9, 9E9, 9E9, 9E9, 9E9, 9E9]];
	VAR robtarget OpenholeUD_5723 := [[481.71, -35.1, 186.75], [0.1589, 0.689022, 0.705057, -0.053802], [0,0,0,0], [9E9, 9E9, 9E9, 9E9, 9E9, 9E9]];
	VAR robtarget OpenholeUD_5724 := [[477.75, -35.1, 186.13], [0.147321, 0.69159, 0.705921, -0.04094], [0,0,0,0], [9E9, 9E9, 9E9, 9E9, 9E9, 9E9]];
	VAR robtarget OpenholeUD_5725 := [[473.8, -35.1, 185.52], [0.135403, 0.694022, 0.706557, -0.027884], [0,0,0,0], [9E9, 9E9, 9E9, 9E9, 9E9, 9E9]];
	VAR robtarget OpenholeUD_5726 := [[469.85, -35.1, 184.91], [0.123166, 0.696297, 0.706955, -0.014668], [0,0,0,0], [9E9, 9E9, 9E9, 9E9, 9E9, 9E9]];
	VAR robtarget OpenholeUD_5727 := [[465.89, -35.1, 184.3], [0.110634, 0.698398, 0.707106, -0.00133], [0,0,0,0], [9E9, 9E9, 9E9, 9E9, 9E9, 9E9]];
	VAR robtarget OpenholeUD_5728 := [[461.94, -35.1, 183.69], [0.097838, 0.700305, 0.707003, 0.012088], [0,0,0,0], [9E9, 9E9, 9E9, 9E9, 9E9, 9E9]];
	VAR robtarget OpenholeUD_5729 := [[457.99, -35.1, 183.08], [0.08481, 0.702002, 0.706645, 0.025545], [0,0,0,0], [9E9, 9E9, 9E9, 9E9, 9E9, 9E9]];
	VAR robtarget OpenholeUD_5730 := [[454.03, -35.1, 182.47], [0.071587, 0.703474, 0.706031, 0.038998], [0,0,0,0], [9E9, 9E9, 9E9, 9E9, 9E9, 9E9]];
	VAR robtarget OpenholeUD_5731 := [[450.08, -35.1, 181.85], [0.058209, 0.704707, 0.705162, 0.052402], [0,0,0,0], [9E9, 9E9, 9E9, 9E9, 9E9, 9E9]];
	VAR robtarget OpenholeUD_5732 := [[446.13, -35.1, 181.24], [0.04472, 0.705691, 0.704047, 0.065715], [0,0,0,0], [9E9, 9E9, 9E9, 9E9, 9E9, 9E9]];
	VAR robtarget OpenholeUD_5733 := [[442.18, -35.1, 180.63], [0.031163, 0.70642, 0.702692, 0.078895], [0,0,0,0], [9E9, 9E9, 9E9, 9E9, 9E9, 9E9]];
	VAR robtarget OpenholeUD_5734 := [[438.22, -35.1, 180.02], [0.017584, 0.706888, 0.701109, 0.091901], [0,0,0,0], [9E9, 9E9, 9E9, 9E9, 9E9, 9E9]];
	VAR robtarget OpenholeUD_5735 := [[434.27, -35.1, 179.41], [0.004027, 0.707095, 0.699313, 0.104697], [0,0,0,0], [9E9, 9E9, 9E9, 9E9, 9E9, 9E9]];
	VAR robtarget OpenholeUD_5736 := [[430.32, -35.1, 178.8], [-0.009463, 0.707043, 0.697318, 0.11725], [0,0,0,0], [9E9, 9E9, 9E9, 9E9, 9E9, 9E9]];
	VAR robtarget OpenholeUD_5737 := [[426.36, -35.1, 178.19], [-0.022843, 0.706738, 0.695142, 0.129527], [0,0,0,0], [9E9, 9E9, 9E9, 9E9, 9E9, 9E9]];
	VAR robtarget OpenholeUD_5738 := [[422.41, -35.1, 177.58], [-0.036073, 0.706186, 0.692803, 0.141505], [0,0,0,0], [9E9, 9E9, 9E9, 9E9, 9E9, 9E9]];
	VAR robtarget OpenholeUD_5739 := [[418.46, -35.1, 176.96], [-0.049116, 0.705399, 0.69032, 0.153159], [0,0,0,0], [9E9, 9E9, 9E9, 9E9, 9E9, 9E9]];
	VAR robtarget OpenholeUD_5740 := [[414.5, -35.1, 176.35], [-0.061938, 0.704389, 0.687712, 0.164473], [0,0,0,0], [9E9, 9E9, 9E9, 9E9, 9E9, 9E9]];
	VAR robtarget OpenholeUD_5741 := [[410.55, -35.1, 175.74], [-0.074509, 0.70317, 0.684999, 0.175433], [0,0,0,0], [9E9, 9E9, 9E9, 9E9, 9E9, 9E9]];
	VAR robtarget OpenholeUD_5742 := [[406.6, -35.1, 175.13], [-0.086803, 0.701759, 0.682197, 0.186029], [0,0,0,0], [9E9, 9E9, 9E9, 9E9, 9E9, 9E9]];
	VAR robtarget OpenholeUD_5743 := [[402.65, -35.1, 174.52], [-0.098798, 0.700171, 0.679326, 0.196254], [0,0,0,0], [9E9, 9E9, 9E9, 9E9, 9E9, 9E9]];
	VAR robtarget OpenholeUD_5744 := [[398.69, -35.1, 173.91], [-0.110476, 0.698423, 0.676402, 0.206107], [0,0,0,0], [9E9, 9E9, 9E9, 9E9, 9E9, 9E9]];
	VAR robtarget OpenholeUD_5745 := [[394.74, -35.1, 173.3], [-0.121824, 0.696534, 0.673441, 0.215586], [0,0,0,0], [9E9, 9E9, 9E9, 9E9, 9E9, 9E9]];
	VAR robtarget OpenholeUD_5746 := [[389.32, -35.1, 172.46], [-0.136831, 0.693742, 0.669345, 0.227986], [0,0,0,0], [9E9, 9E9, 9E9, 9E9, 9E9, 9E9]];
	VAR robtarget OpenholeUD_5747 := [[385.32, -35.1, 172.47], [-0.183051, 0.683002, 0.683002, 0.183051], [0,0,0,0], [9E9, 9E9, 9E9, 9E9, 9E9, 9E9]];
	VAR robtarget OpenholeUD_5748 := [[381.32, -35.1, 172.48], [-0.183051, 0.683002, 0.683002, 0.183051], [0,0,0,0], [9E9, 9E9, 9E9, 9E9, 9E9, 9E9]];
	VAR robtarget OpenholeUD_5749 := [[377.32, -35.1, 172.5], [-0.183051, 0.683002, 0.683002, 0.183051], [0,0,0,0], [9E9, 9E9, 9E9, 9E9, 9E9, 9E9]];
	VAR robtarget OpenholeUD_5750 := [[373.32, -35.1, 172.51], [-0.183051, 0.683002, 0.683002, 0.183051], [0,0,0,0], [9E9, 9E9, 9E9, 9E9, 9E9, 9E9]];
	VAR robtarget OpenholeUD_5751 := [[369.32, -35.1, 172.52], [-0.183051, 0.683002, 0.683002, 0.183051], [0,0,0,0], [9E9, 9E9, 9E9, 9E9, 9E9, 9E9]];
	VAR robtarget OpenholeUD_5752 := [[369.32, -35.1, 172.52], [-0.183051, 0.683002, 0.683002, 0.183051], [0,0,0,0], [9E9, 9E9, 9E9, 9E9, 9E9, 9E9]];
	VAR robtarget OpenholeUD_5753 := [[369.32, -33.9, 173.21], [-0.183051, 0.683002, 0.683002, 0.183051], [0,0,0,0], [9E9, 9E9, 9E9, 9E9, 9E9, 9E9]];
	VAR robtarget OpenholeUD_5754 := [[373.32, -33.9, 173.2], [-0.183051, 0.683002, 0.683002, 0.183051], [0,0,0,0], [9E9, 9E9, 9E9, 9E9, 9E9, 9E9]];
	VAR robtarget OpenholeUD_5755 := [[377.32, -33.9, 173.19], [-0.183051, 0.683002, 0.683002, 0.183051], [0,0,0,0], [9E9, 9E9, 9E9, 9E9, 9E9, 9E9]];
	VAR robtarget OpenholeUD_5756 := [[381.32, -33.9, 173.18], [-0.183051, 0.683002, 0.683002, 0.183051], [0,0,0,0], [9E9, 9E9, 9E9, 9E9, 9E9, 9E9]];
	VAR robtarget OpenholeUD_5757 := [[385.32, -33.9, 173.16], [-0.183051, 0.683002, 0.683002, 0.183051], [0,0,0,0], [9E9, 9E9, 9E9, 9E9, 9E9, 9E9]];
	VAR robtarget OpenholeUD_5758 := [[389.32, -33.9, 173.15], [-0.140254, 0.693058, 0.670457, 0.224695], [0,0,0,0], [9E9, 9E9, 9E9, 9E9, 9E9, 9E9]];
	VAR robtarget OpenholeUD_5759 := [[393.28, -33.9, 173.72], [-0.129422, 0.695162, 0.673424, 0.21564], [0,0,0,0], [9E9, 9E9, 9E9, 9E9, 9E9, 9E9]];
	VAR robtarget OpenholeUD_5760 := [[397.24, -33.9, 174.29], [-0.118243, 0.69715, 0.676369, 0.206217], [0,0,0,0], [9E9, 9E9, 9E9, 9E9, 9E9, 9E9]];
	VAR robtarget OpenholeUD_5761 := [[401.2, -33.9, 174.85], [-0.106726, 0.699006, 0.679278, 0.196421], [0,0,0,0], [9E9, 9E9, 9E9, 9E9, 9E9, 9E9]];
	VAR robtarget OpenholeUD_5762 := [[405.16, -33.9, 175.42], [-0.094883, 0.700712, 0.682136, 0.186253], [0,0,0,0], [9E9, 9E9, 9E9, 9E9, 9E9, 9E9]];
	VAR robtarget OpenholeUD_5763 := [[409.12, -33.9, 175.98], [-0.08273, 0.70225, 0.684927, 0.175714], [0,0,0,0], [9E9, 9E9, 9E9, 9E9, 9E9, 9E9]];
	VAR robtarget OpenholeUD_5764 := [[413.08, -33.9, 176.55], [-0.070287, 0.703605, 0.687632, 0.16481], [0,0,0,0], [9E9, 9E9, 9E9, 9E9, 9E9, 9E9]];
	VAR robtarget OpenholeUD_5765 := [[417.04, -33.9, 177.12], [-0.057578, 0.704759, 0.690234, 0.153549], [0,0,0,0], [9E9, 9E9, 9E9, 9E9, 9E9, 9E9]];
	VAR robtarget OpenholeUD_5766 := [[421, -33.9, 177.68], [-0.044631, 0.705697, 0.692713, 0.141946], [0,0,0,0], [9E9, 9E9, 9E9, 9E9, 9E9, 9E9]];
	VAR robtarget OpenholeUD_5767 := [[424.96, -33.9, 178.25], [-0.031478, 0.706406, 0.695051, 0.130016], [0,0,0,0], [9E9, 9E9, 9E9, 9E9, 9E9, 9E9]];
	VAR robtarget OpenholeUD_5768 := [[428.92, -33.9, 178.82], [-0.018156, 0.706874, 0.697228, 0.117781], [0,0,0,0], [9E9, 9E9, 9E9, 9E9, 9E9, 9E9]];
	VAR robtarget OpenholeUD_5769 := [[432.88, -33.9, 179.38], [-0.004703, 0.707091, 0.699227, 0.105267], [0,0,0,0], [9E9, 9E9, 9E9, 9E9, 9E9, 9E9]];
	VAR robtarget OpenholeUD_5770 := [[436.84, -33.9, 179.95], [0.00884, 0.707052, 0.70103, 0.092502], [0,0,0,0], [9E9, 9E9, 9E9, 9E9, 9E9, 9E9]];
	VAR robtarget OpenholeUD_5771 := [[440.8, -33.9, 180.52], [0.022428, 0.706751, 0.702621, 0.079521], [0,0,0,0], [9E9, 9E9, 9E9, 9E9, 9E9, 9E9]];
	VAR robtarget OpenholeUD_5772 := [[444.76, -33.9, 181.08], [0.036016, 0.706189, 0.703986, 0.066358], [0,0,0,0], [9E9, 9E9, 9E9, 9E9, 9E9, 9E9]];
	VAR robtarget OpenholeUD_5773 := [[448.72, -33.9, 181.65], [0.049559, 0.705368, 0.705114, 0.053055], [0,0,0,0], [9E9, 9E9, 9E9, 9E9, 9E9, 9E9]];
	VAR robtarget OpenholeUD_5774 := [[452.67, -33.9, 182.22], [0.063012, 0.704294, 0.705994, 0.039652], [0,0,0,0], [9E9, 9E9, 9E9, 9E9, 9E9, 9E9]];
	VAR robtarget OpenholeUD_5775 := [[456.63, -33.9, 182.78], [0.076331, 0.702975, 0.706622, 0.026192], [0,0,0,0], [9E9, 9E9, 9E9, 9E9, 9E9, 9E9]];
	VAR robtarget OpenholeUD_5776 := [[460.59, -33.9, 183.35], [0.089475, 0.701423, 0.706992, 0.012719], [0,0,0,0], [9E9, 9E9, 9E9, 9E9, 9E9, 9E9]];
	VAR robtarget OpenholeUD_5777 := [[464.55, -33.9, 183.92], [0.102405, 0.699652, 0.707106, -0.000723], [0,0,0,0], [9E9, 9E9, 9E9, 9E9, 9E9, 9E9]];
	VAR robtarget OpenholeUD_5778 := [[468.51, -33.9, 184.48], [0.115086, 0.697678, 0.706966, -0.014091], [0,0,0,0], [9E9, 9E9, 9E9, 9E9, 9E9, 9E9]];
	VAR robtarget OpenholeUD_5779 := [[472.47, -33.9, 185.05], [0.127487, 0.695519, 0.706578, -0.027345], [0,0,0,0], [9E9, 9E9, 9E9, 9E9, 9E9, 9E9]];
	VAR robtarget OpenholeUD_5780 := [[476.43, -33.9, 185.62], [0.139581, 0.693193, 0.705949, -0.040446], [0,0,0,0], [9E9, 9E9, 9E9, 9E9, 9E9, 9E9]];
	VAR robtarget OpenholeUD_5781 := [[480.39, -33.9, 186.18], [0.151345, 0.69072, 0.705091, -0.053358], [0,0,0,0], [9E9, 9E9, 9E9, 9E9, 9E9, 9E9]];
	VAR robtarget OpenholeUD_5782 := [[484.35, -33.9, 186.75], [0.16276, 0.68812, 0.704015, -0.066049], [0,0,0,0], [9E9, 9E9, 9E9, 9E9, 9E9, 9E9]];
	VAR robtarget OpenholeUD_5783 := [[488.31, -33.9, 187.32], [0.173813, 0.685411, 0.702737, -0.07849], [0,0,0,0], [9E9, 9E9, 9E9, 9E9, 9E9, 9E9]];
	VAR robtarget OpenholeUD_5784 := [[492.27, -33.9, 187.88], [0.184494, 0.682614, 0.701271, -0.090655], [0,0,0,0], [9E9, 9E9, 9E9, 9E9, 9E9, 9E9]];
	VAR robtarget OpenholeUD_5785 := [[496.23, -33.9, 188.45], [0.194797, 0.679746, 0.699635, -0.102525], [0,0,0,0], [9E9, 9E9, 9E9, 9E9, 9E9, 9E9]];
	VAR robtarget OpenholeUD_5786 := [[500.19, -33.9, 189.02], [0.20472, 0.676823, 0.697843, -0.114081], [0,0,0,0], [9E9, 9E9, 9E9, 9E9, 9E9, 9E9]];
	VAR robtarget OpenholeUD_5787 := [[504.15, -33.9, 189.58], [0.214262, 0.673863, 0.695915, -0.125311], [0,0,0,0], [9E9, 9E9, 9E9, 9E9, 9E9, 9E9]];
	VAR robtarget OpenholeUD_5788 := [[509.37, -33.9, 190.33], [0.183051, 0.683002, 0.683002, -0.183051], [0,0,0,0], [9E9, 9E9, 9E9, 9E9, 9E9, 9E9]];
	VAR robtarget OpenholeUD_5789 := [[513.37, -33.9, 190.32], [0.183051, 0.683002, 0.683002, -0.183051], [0,0,0,0], [9E9, 9E9, 9E9, 9E9, 9E9, 9E9]];
	VAR robtarget OpenholeUD_5790 := [[517.37, -33.9, 190.31], [0.183051, 0.683002, 0.683002, -0.183051], [0,0,0,0], [9E9, 9E9, 9E9, 9E9, 9E9, 9E9]];
	VAR robtarget OpenholeUD_5791 := [[521.37, -33.9, 190.29], [0.183051, 0.683002, 0.683002, -0.183051], [0,0,0,0], [9E9, 9E9, 9E9, 9E9, 9E9, 9E9]];
	VAR robtarget OpenholeUD_5792 := [[525.37, -33.9, 190.28], [0.183051, 0.683002, 0.683002, -0.183051], [0,0,0,0], [9E9, 9E9, 9E9, 9E9, 9E9, 9E9]];
	VAR robtarget OpenholeUD_5793 := [[529.37, -33.9, 190.27], [0.183051, 0.683002, 0.683002, -0.183051], [0,0,0,0], [9E9, 9E9, 9E9, 9E9, 9E9, 9E9]];
	VAR robtarget OpenholeUD_5794 := [[529.37, -33.9, 190.27], [0.183051, 0.683002, 0.683002, -0.183051], [0,0,0,0], [9E9, 9E9, 9E9, 9E9, 9E9, 9E9]];
	VAR robtarget OpenholeUD_5795 := [[529.37, -32.7, 189.58], [0.183051, 0.683002, 0.683002, -0.183051], [0,0,0,0], [9E9, 9E9, 9E9, 9E9, 9E9, 9E9]];
	VAR robtarget OpenholeUD_5796 := [[525.37, -32.7, 189.59], [0.183051, 0.683002, 0.683002, -0.183051], [0,0,0,0], [9E9, 9E9, 9E9, 9E9, 9E9, 9E9]];
	VAR robtarget OpenholeUD_5797 := [[521.37, -32.7, 189.6], [0.183051, 0.683002, 0.683002, -0.183051], [0,0,0,0], [9E9, 9E9, 9E9, 9E9, 9E9, 9E9]];
	VAR robtarget OpenholeUD_5798 := [[517.37, -32.7, 189.61], [0.183051, 0.683002, 0.683002, -0.183051], [0,0,0,0], [9E9, 9E9, 9E9, 9E9, 9E9, 9E9]];
	VAR robtarget OpenholeUD_5799 := [[509.37, -32.7, 189.64], [0.183051, 0.683002, 0.683002, -0.183051], [0,0,0,0], [9E9, 9E9, 9E9, 9E9, 9E9, 9E9]];
	VAR robtarget OpenholeUD_5800 := [[505.41, -32.7, 189.12], [0.213838, 0.673998, 0.694625, -0.132272], [0,0,0,0], [9E9, 9E9, 9E9, 9E9, 9E9, 9E9]];
	VAR robtarget OpenholeUD_5801 := [[501.44, -32.7, 188.59], [0.204333, 0.67694, 0.696644, -0.121193], [0,0,0,0], [9E9, 9E9, 9E9, 9E9, 9E9, 9E9]];
	VAR robtarget OpenholeUD_5802 := [[497.48, -32.7, 188.07], [0.194449, 0.679845, 0.698533, -0.10978], [0,0,0,0], [9E9, 9E9, 9E9, 9E9, 9E9, 9E9]];
	VAR robtarget OpenholeUD_5803 := [[493.51, -32.7, 187.55], [0.184186, 0.682697, 0.700276, -0.098047], [0,0,0,0], [9E9, 9E9, 9E9, 9E9, 9E9, 9E9]];
	VAR robtarget OpenholeUD_5804 := [[489.54, -32.7, 187.03], [0.173544, 0.68548, 0.701857, -0.086007], [0,0,0,0], [9E9, 9E9, 9E9, 9E9, 9E9, 9E9]];
	VAR robtarget OpenholeUD_5805 := [[485.58, -32.7, 186.51], [0.162529, 0.688175, 0.703257, -0.073681], [0,0,0,0], [9E9, 9E9, 9E9, 9E9, 9E9, 9E9]];
	VAR robtarget OpenholeUD_5806 := [[481.61, -32.7, 185.99], [0.15115, 0.690763, 0.704463, -0.061092], [0,0,0,0], [9E9, 9E9, 9E9, 9E9, 9E9, 9E9]];
	VAR robtarget OpenholeUD_5807 := [[477.65, -32.7, 185.46], [0.139422, 0.693225, 0.705457, -0.048268], [0,0,0,0], [9E9, 9E9, 9E9, 9E9, 9E9, 9E9]];
	VAR robtarget OpenholeUD_5808 := [[473.68, -32.7, 184.94], [0.127361, 0.695542, 0.706228, -0.035238], [0,0,0,0], [9E9, 9E9, 9E9, 9E9, 9E9, 9E9]];
	VAR robtarget OpenholeUD_5809 := [[469.71, -32.7, 184.42], [0.114989, 0.697694, 0.706763, -0.022038], [0,0,0,0], [9E9, 9E9, 9E9, 9E9, 9E9, 9E9]];
	VAR robtarget OpenholeUD_5810 := [[465.75, -32.7, 183.9], [0.102332, 0.699663, 0.707053, -0.008705], [0,0,0,0], [9E9, 9E9, 9E9, 9E9, 9E9, 9E9]];
	VAR robtarget OpenholeUD_5811 := [[461.78, -32.7, 183.38], [0.089422, 0.70143, 0.707091, 0.004721], [0,0,0,0], [9E9, 9E9, 9E9, 9E9, 9E9, 9E9]];
	VAR robtarget OpenholeUD_5812 := [[457.82, -32.7, 182.86], [0.076293, 0.702979, 0.706873, 0.018196], [0,0,0,0], [9E9, 9E9, 9E9, 9E9, 9E9, 9E9]];
	VAR robtarget OpenholeUD_5813 := [[453.85, -32.7, 182.33], [0.062983, 0.704296, 0.706397, 0.031679], [0,0,0,0], [9E9, 9E9, 9E9, 9E9, 9E9, 9E9]];
	VAR robtarget OpenholeUD_5814 := [[449.89, -32.7, 181.81], [0.049534, 0.70537, 0.705665, 0.045125], [0,0,0,0], [9E9, 9E9, 9E9, 9E9, 9E9, 9E9]];
	VAR robtarget OpenholeUD_5815 := [[445.92, -32.7, 181.29], [0.035987, 0.70619, 0.704683, 0.058491], [0,0,0,0], [9E9, 9E9, 9E9, 9E9, 9E9, 9E9]];
	VAR robtarget OpenholeUD_5816 := [[441.95, -32.7, 180.77], [0.02239, 0.706752, 0.703459, 0.071734], [0,0,0,0], [9E9, 9E9, 9E9, 9E9, 9E9, 9E9]];
	VAR robtarget OpenholeUD_5817 := [[437.99, -32.7, 180.25], [0.008786, 0.707052, 0.702002, 0.084813], [0,0,0,0], [9E9, 9E9, 9E9, 9E9, 9E9, 9E9]];
	VAR robtarget OpenholeUD_5818 := [[434.02, -32.7, 179.73], [-0.004778, 0.707091, 0.700326, 0.097692], [0,0,0,0], [9E9, 9E9, 9E9, 9E9, 9E9, 9E9]];
	VAR robtarget OpenholeUD_5819 := [[430.06, -32.7, 179.2], [-0.018258, 0.706871, 0.698446, 0.110334], [0,0,0,0], [9E9, 9E9, 9E9, 9E9, 9E9, 9E9]];
	VAR robtarget OpenholeUD_5820 := [[426.09, -32.7, 178.68], [-0.031613, 0.7064, 0.696378, 0.12271], [0,0,0,0], [9E9, 9E9, 9E9, 9E9, 9E9, 9E9]];
	VAR robtarget OpenholeUD_5821 := [[422.12, -32.7, 178.16], [-0.044802, 0.705686, 0.694141, 0.134792], [0,0,0,0], [9E9, 9E9, 9E9, 9E9, 9E9, 9E9]];
	VAR robtarget OpenholeUD_5822 := [[418.16, -32.7, 177.64], [-0.057789, 0.704741, 0.691752, 0.146557], [0,0,0,0], [9E9, 9E9, 9E9, 9E9, 9E9, 9E9]];
	VAR robtarget OpenholeUD_5823 := [[414.19, -32.7, 177.12], [-0.070542, 0.703579, 0.689232, 0.157986], [0,0,0,0], [9E9, 9E9, 9E9, 9E9, 9E9, 9E9]];
	VAR robtarget OpenholeUD_5824 := [[410.23, -32.7, 176.6], [-0.083031, 0.702215, 0.686598, 0.169064], [0,0,0,0], [9E9, 9E9, 9E9, 9E9, 9E9, 9E9]];
	VAR robtarget OpenholeUD_5825 := [[406.26, -32.7, 176.07], [-0.095231, 0.700665, 0.68387, 0.179782], [0,0,0,0], [9E9, 9E9, 9E9, 9E9, 9E9, 9E9]];
	VAR robtarget OpenholeUD_5826 := [[402.3, -32.7, 175.55], [-0.107122, 0.698946, 0.681065, 0.190131], [0,0,0,0], [9E9, 9E9, 9E9, 9E9, 9E9, 9E9]];
	VAR robtarget OpenholeUD_5827 := [[398.33, -32.7, 175.03], [-0.118687, 0.697075, 0.678201, 0.200109], [0,0,0,0], [9E9, 9E9, 9E9, 9E9, 9E9, 9E9]];
	VAR robtarget OpenholeUD_5828 := [[394.36, -32.7, 174.51], [-0.129913, 0.69507, 0.675292, 0.209715], [0,0,0,0], [9E9, 9E9, 9E9, 9E9, 9E9, 9E9]];
	VAR robtarget OpenholeUD_5829 := [[389.32, -32.7, 173.84], [-0.143682, 0.692355, 0.671555, 0.221391], [0,0,0,0], [9E9, 9E9, 9E9, 9E9, 9E9, 9E9]];
	VAR robtarget OpenholeUD_5830 := [[385.32, -32.7, 173.86], [-0.183051, 0.683002, 0.683002, 0.183051], [0,0,0,0], [9E9, 9E9, 9E9, 9E9, 9E9, 9E9]];
	VAR robtarget OpenholeUD_5831 := [[381.32, -32.7, 173.87], [-0.183051, 0.683002, 0.683002, 0.183051], [0,0,0,0], [9E9, 9E9, 9E9, 9E9, 9E9, 9E9]];
	VAR robtarget OpenholeUD_5832 := [[377.32, -32.7, 173.88], [-0.183051, 0.683002, 0.683002, 0.183051], [0,0,0,0], [9E9, 9E9, 9E9, 9E9, 9E9, 9E9]];
	VAR robtarget OpenholeUD_5833 := [[373.32, -32.7, 173.9], [-0.183051, 0.683002, 0.683002, 0.183051], [0,0,0,0], [9E9, 9E9, 9E9, 9E9, 9E9, 9E9]];
	VAR robtarget OpenholeUD_5834 := [[369.32, -32.7, 173.91], [-0.183051, 0.683002, 0.683002, 0.183051], [0,0,0,0], [9E9, 9E9, 9E9, 9E9, 9E9, 9E9]];
	VAR robtarget OpenholeUD_5835 := [[369.32, -32.7, 173.91], [-0.183051, 0.683002, 0.683002, 0.183051], [0,0,0,0], [9E9, 9E9, 9E9, 9E9, 9E9, 9E9]];
	VAR robtarget OpenholeUD_5836 := [[369.32, -31.5, 174.6], [-0.183051, 0.683002, 0.683002, 0.183051], [0,0,0,0], [9E9, 9E9, 9E9, 9E9, 9E9, 9E9]];
	VAR robtarget OpenholeUD_5837 := [[373.32, -31.5, 174.59], [-0.183051, 0.683002, 0.683002, 0.183051], [0,0,0,0], [9E9, 9E9, 9E9, 9E9, 9E9, 9E9]];
	VAR robtarget OpenholeUD_5838 := [[377.32, -31.5, 174.58], [-0.183051, 0.683002, 0.683002, 0.183051], [0,0,0,0], [9E9, 9E9, 9E9, 9E9, 9E9, 9E9]];
	VAR robtarget OpenholeUD_5839 := [[381.32, -31.5, 174.56], [-0.183051, 0.683002, 0.683002, 0.183051], [0,0,0,0], [9E9, 9E9, 9E9, 9E9, 9E9, 9E9]];
	VAR robtarget OpenholeUD_5840 := [[385.32, -31.5, 174.55], [-0.183051, 0.683002, 0.683002, 0.183051], [0,0,0,0], [9E9, 9E9, 9E9, 9E9, 9E9, 9E9]];
	VAR robtarget OpenholeUD_5841 := [[389.32, -31.5, 174.54], [-0.147114, 0.691634, 0.672639, 0.218075], [0,0,0,0], [9E9, 9E9, 9E9, 9E9, 9E9, 9E9]];
	VAR robtarget OpenholeUD_5842 := [[393.3, -31.5, 175.01], [-0.13638, 0.69383, 0.675558, 0.208858], [0,0,0,0], [9E9, 9E9, 9E9, 9E9, 9E9, 9E9]];
	VAR robtarget OpenholeUD_5843 := [[397.27, -31.5, 175.49], [-0.125295, 0.695918, 0.678447, 0.199272], [0,0,0,0], [9E9, 9E9, 9E9, 9E9, 9E9, 9E9]];
	VAR robtarget OpenholeUD_5844 := [[401.24, -31.5, 175.97], [-0.113865, 0.697879, 0.681293, 0.189315], [0,0,0,0], [9E9, 9E9, 9E9, 9E9, 9E9, 9E9]];
	VAR robtarget OpenholeUD_5845 := [[405.21, -31.5, 176.44], [-0.102102, 0.699696, 0.684079, 0.178987], [0,0,0,0], [9E9, 9E9, 9E9, 9E9, 9E9, 9E9]];
	VAR robtarget OpenholeUD_5846 := [[409.18, -31.5, 176.92], [-0.090022, 0.701353, 0.686788, 0.16829], [0,0,0,0], [9E9, 9E9, 9E9, 9E9, 9E9, 9E9]];
	VAR robtarget OpenholeUD_5847 := [[413.15, -31.5, 177.4], [-0.077642, 0.702831, 0.689404, 0.157233], [0,0,0,0], [9E9, 9E9, 9E9, 9E9, 9E9, 9E9]];
	VAR robtarget OpenholeUD_5848 := [[417.13, -31.5, 177.87], [-0.064986, 0.704114, 0.691907, 0.145824], [0,0,0,0], [9E9, 9E9, 9E9, 9E9, 9E9, 9E9]];
	VAR robtarget OpenholeUD_5849 := [[421.1, -31.5, 178.35], [-0.052082, 0.705186, 0.694279, 0.134078], [0,0,0,0], [9E9, 9E9, 9E9, 9E9, 9E9, 9E9]];
	VAR robtarget OpenholeUD_5850 := [[425.07, -31.5, 178.83], [-0.038962, 0.706033, 0.6965, 0.122013], [0,0,0,0], [9E9, 9E9, 9E9, 9E9, 9E9, 9E9]];
	VAR robtarget OpenholeUD_5851 := [[429.04, -31.5, 179.3], [-0.025659, 0.706641, 0.698553, 0.109653], [0,0,0,0], [9E9, 9E9, 9E9, 9E9, 9E9, 9E9]];
	VAR robtarget OpenholeUD_5852 := [[433.01, -31.5, 179.78], [-0.012214, 0.707001, 0.700419, 0.097023], [0,0,0,0], [9E9, 9E9, 9E9, 9E9, 9E9, 9E9]];
	VAR robtarget OpenholeUD_5853 := [[436.98, -31.5, 180.26], [0.001333, 0.707106, 0.702081, 0.084154], [0,0,0,0], [9E9, 9E9, 9E9, 9E9, 9E9, 9E9]];
	VAR robtarget OpenholeUD_5854 := [[440.95, -31.5, 180.73], [0.014937, 0.706949, 0.703525, 0.071081], [0,0,0,0], [9E9, 9E9, 9E9, 9E9, 9E9, 9E9]];
	VAR robtarget OpenholeUD_5855 := [[444.93, -31.5, 181.21], [0.028555, 0.70653, 0.704737, 0.057841], [0,0,0,0], [9E9, 9E9, 9E9, 9E9, 9E9, 9E9]];
	VAR robtarget OpenholeUD_5856 := [[448.9, -31.5, 181.69], [0.042139, 0.70585, 0.705707, 0.044474], [0,0,0,0], [9E9, 9E9, 9E9, 9E9, 9E9, 9E9]];
	VAR robtarget OpenholeUD_5857 := [[452.87, -31.5, 182.16], [0.055645, 0.704914, 0.706426, 0.031023], [0,0,0,0], [9E9, 9E9, 9E9, 9E9, 9E9, 9E9]];
	VAR robtarget OpenholeUD_5858 := [[456.84, -31.5, 182.64], [0.069029, 0.703729, 0.706889, 0.017531], [0,0,0,0], [9E9, 9E9, 9E9, 9E9, 9E9, 9E9]];
	VAR robtarget OpenholeUD_5859 := [[460.81, -31.5, 183.12], [0.082248, 0.702307, 0.707095, 0.004042], [0,0,0,0], [9E9, 9E9, 9E9, 9E9, 9E9, 9E9]];
	VAR robtarget OpenholeUD_5860 := [[464.78, -31.5, 183.59], [0.095262, 0.70066, 0.707044, -0.0094], [0,0,0,0], [9E9, 9E9, 9E9, 9E9, 9E9, 9E9]];
	VAR robtarget OpenholeUD_5861 := [[468.75, -31.5, 184.07], [0.108037, 0.698805, 0.706741, -0.022754], [0,0,0,0], [9E9, 9E9, 9E9, 9E9, 9E9, 9E9]];
	VAR robtarget OpenholeUD_5862 := [[472.73, -31.5, 184.55], [0.120539, 0.696757, 0.706191, -0.035977], [0,0,0,0], [9E9, 9E9, 9E9, 9E9, 9E9, 9E9]];
	VAR robtarget OpenholeUD_5863 := [[476.7, -31.5, 185.02], [0.132741, 0.694536, 0.705405, -0.049033], [0,0,0,0], [9E9, 9E9, 9E9, 9E9, 9E9, 9E9]];
	VAR robtarget OpenholeUD_5864 := [[480.67, -31.5, 185.5], [0.144619, 0.69216, 0.704393, -0.061886], [0,0,0,0], [9E9, 9E9, 9E9, 9E9, 9E9, 9E9]];
	VAR robtarget OpenholeUD_5865 := [[484.64, -31.5, 185.98], [0.156153, 0.689649, 0.703171, -0.074504], [0,0,0,0], [9E9, 9E9, 9E9, 9E9, 9E9, 9E9]];
	VAR robtarget OpenholeUD_5866 := [[488.61, -31.5, 186.45], [0.167329, 0.687023, 0.701751, -0.086861], [0,0,0,0], [9E9, 9E9, 9E9, 9E9, 9E9, 9E9]];
	VAR robtarget OpenholeUD_5867 := [[492.58, -31.5, 186.93], [0.178136, 0.684301, 0.700152, -0.098932], [0,0,0,0], [9E9, 9E9, 9E9, 9E9, 9E9, 9E9]];
	VAR robtarget OpenholeUD_5868 := [[496.56, -31.5, 187.41], [0.188567, 0.6815, 0.698388, -0.110697], [0,0,0,0], [9E9, 9E9, 9E9, 9E9, 9E9, 9E9]];
	VAR robtarget OpenholeUD_5869 := [[500.53, -31.5, 187.88], [0.198619, 0.678639, 0.696478, -0.122141], [0,0,0,0], [9E9, 9E9, 9E9, 9E9, 9E9, 9E9]];
	VAR robtarget OpenholeUD_5870 := [[504.5, -31.5, 188.36], [0.208291, 0.675733, 0.694438, -0.133251], [0,0,0,0], [9E9, 9E9, 9E9, 9E9, 9E9, 9E9]];
	VAR robtarget OpenholeUD_5871 := [[509.37, -31.5, 188.94], [0.183051, 0.683002, 0.683002, -0.183051], [0,0,0,0], [9E9, 9E9, 9E9, 9E9, 9E9, 9E9]];
	VAR robtarget OpenholeUD_5872 := [[513.37, -31.5, 188.93], [0.183051, 0.683002, 0.683002, -0.183051], [0,0,0,0], [9E9, 9E9, 9E9, 9E9, 9E9, 9E9]];
	VAR robtarget OpenholeUD_5873 := [[517.37, -31.5, 188.92], [0.183051, 0.683002, 0.683002, -0.183051], [0,0,0,0], [9E9, 9E9, 9E9, 9E9, 9E9, 9E9]];
	VAR robtarget OpenholeUD_5874 := [[521.37, -31.5, 188.91], [0.183051, 0.683002, 0.683002, -0.183051], [0,0,0,0], [9E9, 9E9, 9E9, 9E9, 9E9, 9E9]];
	VAR robtarget OpenholeUD_5875 := [[525.37, -31.5, 188.89], [0.183051, 0.683002, 0.683002, -0.183051], [0,0,0,0], [9E9, 9E9, 9E9, 9E9, 9E9, 9E9]];
	VAR robtarget OpenholeUD_5876 := [[529.37, -31.5, 188.88], [0.183051, 0.683002, 0.683002, -0.183051], [0,0,0,0], [9E9, 9E9, 9E9, 9E9, 9E9, 9E9]];
	VAR robtarget OpenholeUD_5877 := [[529.37, -31.5, 188.88], [0.183051, 0.683002, 0.683002, -0.183051], [0,0,0,0], [9E9, 9E9, 9E9, 9E9, 9E9, 9E9]];
	VAR robtarget OpenholeUD_5878 := [[529.37, -30.3, 188.19], [0.183051, 0.683002, 0.683002, -0.183051], [0,0,0,0], [9E9, 9E9, 9E9, 9E9, 9E9, 9E9]];
	VAR robtarget OpenholeUD_5879 := [[525.37, -30.3, 188.2], [0.183051, 0.683002, 0.683002, -0.183051], [0,0,0,0], [9E9, 9E9, 9E9, 9E9, 9E9, 9E9]];
	VAR robtarget OpenholeUD_5880 := [[521.37, -30.3, 188.21], [0.183051, 0.683002, 0.683002, -0.183051], [0,0,0,0], [9E9, 9E9, 9E9, 9E9, 9E9, 9E9]];
	VAR robtarget OpenholeUD_5881 := [[517.37, -30.3, 188.23], [0.183051, 0.683002, 0.683002, -0.183051], [0,0,0,0], [9E9, 9E9, 9E9, 9E9, 9E9, 9E9]];
	VAR robtarget OpenholeUD_5882 := [[513.37, -30.3, 188.24], [0.183051, 0.683002, 0.683002, -0.183051], [0,0,0,0], [9E9, 9E9, 9E9, 9E9, 9E9, 9E9]];
	VAR robtarget OpenholeUD_5883 := [[509.37, -30.3, 188.25], [0.183051, 0.683002, 0.683002, -0.183051], [0,0,0,0], [9E9, 9E9, 9E9, 9E9, 9E9, 9E9]];
	VAR robtarget OpenholeUD_5884 := [[505.39, -30.3, 187.82], [0.207015, 0.676125, 0.693274, -0.139181], [0,0,0,0], [9E9, 9E9, 9E9, 9E9, 9E9, 9E9]];
	VAR robtarget OpenholeUD_5885 := [[501.41, -30.3, 187.39], [0.197347, 0.67901, 0.695389, -0.128196], [0,0,0,0], [9E9, 9E9, 9E9, 9E9, 9E9, 9E9]];
	VAR robtarget OpenholeUD_5886 := [[497.44, -30.3, 186.96], [0.1873, 0.681849, 0.697381, -0.116873], [0,0,0,0], [9E9, 9E9, 9E9, 9E9, 9E9, 9E9]];
	VAR robtarget OpenholeUD_5887 := [[493.46, -30.3, 186.53], [0.176875, 0.684628, 0.699234, -0.105222], [0,0,0,0], [9E9, 9E9, 9E9, 9E9, 9E9, 9E9]];
	VAR robtarget OpenholeUD_5888 := [[489.48, -30.3, 186.1], [0.166073, 0.687328, 0.70093, -0.093257], [0,0,0,0], [9E9, 9E9, 9E9, 9E9, 9E9, 9E9]];
	VAR robtarget OpenholeUD_5889 := [[485.51, -30.3, 185.66], [0.154904, 0.689931, 0.702452, -0.080998], [0,0,0,0], [9E9, 9E9, 9E9, 9E9, 9E9, 9E9]];
	VAR robtarget OpenholeUD_5890 := [[481.53, -30.3, 185.23], [0.143375, 0.692419, 0.703784, -0.068467], [0,0,0,0], [9E9, 9E9, 9E9, 9E9, 9E9, 9E9]];
	VAR robtarget OpenholeUD_5891 := [[477.55, -30.3, 184.8], [0.131503, 0.694771, 0.70491, -0.055689], [0,0,0,0], [9E9, 9E9, 9E9, 9E9, 9E9, 9E9]];
	VAR robtarget OpenholeUD_5892 := [[473.58, -30.3, 184.37], [0.119306, 0.696969, 0.705817, -0.042696], [0,0,0,0], [9E9, 9E9, 9E9, 9E9, 9E9, 9E9]];
	VAR robtarget OpenholeUD_5893 := [[469.6, -30.3, 183.94], [0.106807, 0.698994, 0.70649, -0.029521], [0,0,0,0], [9E9, 9E9, 9E9, 9E9, 9E9, 9E9]];
	VAR robtarget OpenholeUD_5894 := [[465.62, -30.3, 183.51], [0.094034, 0.700826, 0.706921, -0.016202], [0,0,0,0], [9E9, 9E9, 9E9, 9E9, 9E9, 9E9]];
	VAR robtarget OpenholeUD_5895 := [[461.65, -30.3, 183.08], [0.08102, 0.70245, 0.707101, -0.002778], [0,0,0,0], [9E9, 9E9, 9E9, 9E9, 9E9, 9E9]];
	VAR robtarget OpenholeUD_5896 := [[457.67, -30.3, 182.64], [0.067799, 0.703849, 0.707026, 0.010709], [0,0,0,0], [9E9, 9E9, 9E9, 9E9, 9E9, 9E9]];
	VAR robtarget OpenholeUD_5897 := [[453.69, -30.3, 182.21], [0.054412, 0.70501, 0.706692, 0.024214], [0,0,0,0], [9E9, 9E9, 9E9, 9E9, 9E9, 9E9]];
	VAR robtarget OpenholeUD_5898 := [[449.72, -30.3, 181.78], [0.040901, 0.705923, 0.706101, 0.037695], [0,0,0,0], [9E9, 9E9, 9E9, 9E9, 9E9, 9E9]];
	VAR robtarget OpenholeUD_5899 := [[445.74, -30.3, 181.35], [0.027308, 0.706579, 0.705257, 0.051108], [0,0,0,0], [9E9, 9E9, 9E9, 9E9, 9E9, 9E9]];
	VAR robtarget OpenholeUD_5900 := [[441.76, -30.3, 180.92], [0.013681, 0.706974, 0.704167, 0.064408], [0,0,0,0], [9E9, 9E9, 9E9, 9E9, 9E9, 9E9]];
	VAR robtarget OpenholeUD_5901 := [[437.79, -30.3, 180.49], [0.000064, 0.707107, 0.702841, 0.077557], [0,0,0,0], [9E9, 9E9, 9E9, 9E9, 9E9, 9E9]];
	VAR robtarget OpenholeUD_5902 := [[433.81, -30.3, 180.06], [-0.013497, 0.706978, 0.70129, 0.090514], [0,0,0,0], [9E9, 9E9, 9E9, 9E9, 9E9, 9E9]];
	VAR robtarget OpenholeUD_5903 := [[429.83, -30.3, 179.62], [-0.026958, 0.706593, 0.699529, 0.103244], [0,0,0,0], [9E9, 9E9, 9E9, 9E9, 9E9, 9E9]];
	VAR robtarget OpenholeUD_5904 := [[425.86, -30.3, 179.19], [-0.040277, 0.705959, 0.697574, 0.115716], [0,0,0,0], [9E9, 9E9, 9E9, 9E9, 9E9, 9E9]];
	VAR robtarget OpenholeUD_5905 := [[421.88, -30.3, 178.76], [-0.053416, 0.705086, 0.695443, 0.127901], [0,0,0,0], [9E9, 9E9, 9E9, 9E9, 9E9, 9E9]];
	VAR robtarget OpenholeUD_5906 := [[417.9, -30.3, 178.33], [-0.066338, 0.703988, 0.693154, 0.139776], [0,0,0,0], [9E9, 9E9, 9E9, 9E9, 9E9, 9E9]];
	VAR robtarget OpenholeUD_5907 := [[413.93, -30.3, 177.9], [-0.079013, 0.702678, 0.690726, 0.151321], [0,0,0,0], [9E9, 9E9, 9E9, 9E9, 9E9, 9E9]];
	VAR robtarget OpenholeUD_5908 := [[409.95, -30.3, 177.47], [-0.091411, 0.701173, 0.688177, 0.162519], [0,0,0,0], [9E9, 9E9, 9E9, 9E9, 9E9, 9E9]];
	VAR robtarget OpenholeUD_5909 := [[405.97, -30.3, 177.04], [-0.10351, 0.69949, 0.685526, 0.17336], [0,0,0,0], [9E9, 9E9, 9E9, 9E9, 9E9, 9E9]];
	VAR robtarget OpenholeUD_5910 := [[402, -30.3, 176.61], [-0.115291, 0.697645, 0.682792, 0.183836], [0,0,0,0], [9E9, 9E9, 9E9, 9E9, 9E9, 9E9]];
	VAR robtarget OpenholeUD_5911 := [[398.02, -30.3, 176.17], [-0.126737, 0.695656, 0.67999, 0.193941], [0,0,0,0], [9E9, 9E9, 9E9, 9E9, 9E9, 9E9]];
	VAR robtarget OpenholeUD_5912 := [[394.04, -30.3, 175.74], [-0.137838, 0.693542, 0.677138, 0.203676], [0,0,0,0], [9E9, 9E9, 9E9, 9E9, 9E9, 9E9]];
	VAR robtarget OpenholeUD_5913 := [[389.33, -30.3, 175.23], [-0.150549, 0.690894, 0.673709, 0.214746], [0,0,0,0], [9E9, 9E9, 9E9, 9E9, 9E9, 9E9]];
	VAR robtarget OpenholeUD_5914 := [[385.33, -30.3, 175.24], [-0.183051, 0.683002, 0.683002, 0.183051], [0,0,0,0], [9E9, 9E9, 9E9, 9E9, 9E9, 9E9]];
	VAR robtarget OpenholeUD_5915 := [[381.33, -30.3, 175.26], [-0.183051, 0.683002, 0.683002, 0.183051], [0,0,0,0], [9E9, 9E9, 9E9, 9E9, 9E9, 9E9]];
	VAR robtarget OpenholeUD_5916 := [[377.33, -30.3, 175.27], [-0.183051, 0.683002, 0.683002, 0.183051], [0,0,0,0], [9E9, 9E9, 9E9, 9E9, 9E9, 9E9]];
	VAR robtarget OpenholeUD_5917 := [[373.33, -30.3, 175.28], [-0.183051, 0.683002, 0.683002, 0.183051], [0,0,0,0], [9E9, 9E9, 9E9, 9E9, 9E9, 9E9]];
	VAR robtarget OpenholeUD_5918 := [[369.33, -30.3, 175.29], [-0.183051, 0.683002, 0.683002, 0.183051], [0,0,0,0], [9E9, 9E9, 9E9, 9E9, 9E9, 9E9]];
	VAR robtarget OpenholeUD_5919 := [[369.33, -30.3, 175.29], [-0.183051, 0.683002, 0.683002, 0.183051], [0,0,0,0], [9E9, 9E9, 9E9, 9E9, 9E9, 9E9]];
	VAR robtarget OpenholeUD_5920 := [[369.33, -29.1, 175.99], [-0.183051, 0.683002, 0.683002, 0.183051], [0,0,0,0], [9E9, 9E9, 9E9, 9E9, 9E9, 9E9]];
	VAR robtarget OpenholeUD_5921 := [[373.33, -29.1, 175.97], [-0.183051, 0.683002, 0.683002, 0.183051], [0,0,0,0], [9E9, 9E9, 9E9, 9E9, 9E9, 9E9]];
	VAR robtarget OpenholeUD_5922 := [[377.33, -29.1, 175.96], [-0.183051, 0.683002, 0.683002, 0.183051], [0,0,0,0], [9E9, 9E9, 9E9, 9E9, 9E9, 9E9]];
	VAR robtarget OpenholeUD_5923 := [[381.33, -29.1, 175.95], [-0.183051, 0.683002, 0.683002, 0.183051], [0,0,0,0], [9E9, 9E9, 9E9, 9E9, 9E9, 9E9]];
	VAR robtarget OpenholeUD_5924 := [[385.33, -29.1, 175.94], [-0.183051, 0.683002, 0.683002, 0.183051], [0,0,0,0], [9E9, 9E9, 9E9, 9E9, 9E9, 9E9]];
	VAR robtarget OpenholeUD_5925 := [[389.33, -29.1, 175.92], [-0.153987, 0.690136, 0.674765, 0.211407], [0,0,0,0], [9E9, 9E9, 9E9, 9E9, 9E9, 9E9]];
	VAR robtarget OpenholeUD_5926 := [[393.31, -29.1, 176.31], [-0.143361, 0.692422, 0.677631, 0.202031], [0,0,0,0], [9E9, 9E9, 9E9, 9E9, 9E9, 9E9]];
	VAR robtarget OpenholeUD_5927 := [[397.29, -29.1, 176.7], [-0.132377, 0.694605, 0.68046, 0.192286], [0,0,0,0], [9E9, 9E9, 9E9, 9E9, 9E9, 9E9]];
	VAR robtarget OpenholeUD_5928 := [[401.27, -29.1, 177.08], [-0.121044, 0.696669, 0.683238, 0.182171], [0,0,0,0], [9E9, 9E9, 9E9, 9E9, 9E9, 9E9]];
	VAR robtarget OpenholeUD_5929 := [[405.25, -29.1, 177.47], [-0.109371, 0.698597, 0.685947, 0.171687], [0,0,0,0], [9E9, 9E9, 9E9, 9E9, 9E9, 9E9]];
	VAR robtarget OpenholeUD_5930 := [[409.24, -29.1, 177.85], [-0.097372, 0.70037, 0.688572, 0.160838], [0,0,0,0], [9E9, 9E9, 9E9, 9E9, 9E9, 9E9]];
	VAR robtarget OpenholeUD_5931 := [[413.22, -29.1, 178.24], [-0.085066, 0.701971, 0.691094, 0.149632], [0,0,0,0], [9E9, 9E9, 9E9, 9E9, 9E9, 9E9]];
	VAR robtarget OpenholeUD_5932 := [[417.2, -29.1, 178.63], [-0.072474, 0.703383, 0.693494, 0.138081], [0,0,0,0], [9E9, 9E9, 9E9, 9E9, 9E9, 9E9]];
	VAR robtarget OpenholeUD_5933 := [[421.18, -29.1, 179.01], [-0.059623, 0.704589, 0.695754, 0.126199], [0,0,0,0], [9E9, 9E9, 9E9, 9E9, 9E9, 9E9]];
	VAR robtarget OpenholeUD_5934 := [[425.16, -29.1, 179.4], [-0.046544, 0.705573, 0.697856, 0.114007], [0,0,0,0], [9E9, 9E9, 9E9, 9E9, 9E9, 9E9]];
	VAR robtarget OpenholeUD_5935 := [[429.14, -29.1, 179.78], [-0.033272, 0.706324, 0.69978, 0.101529], [0,0,0,0], [9E9, 9E9, 9E9, 9E9, 9E9, 9E9]];
	VAR robtarget OpenholeUD_5936 := [[433.12, -29.1, 180.17], [-0.019845, 0.706828, 0.70151, 0.088791], [0,0,0,0], [9E9, 9E9, 9E9, 9E9, 9E9, 9E9]];
	VAR robtarget OpenholeUD_5937 := [[437.11, -29.1, 180.55], [-0.006303, 0.707079, 0.703029, 0.075828], [0,0,0,0], [9E9, 9E9, 9E9, 9E9, 9E9, 9E9]];
	VAR robtarget OpenholeUD_5938 := [[441.09, -29.1, 180.94], [0.00731, 0.707069, 0.704324, 0.062672], [0,0,0,0], [9E9, 9E9, 9E9, 9E9, 9E9, 9E9]];
	VAR robtarget OpenholeUD_5939 := [[445.07, -29.1, 181.33], [0.020948, 0.706796, 0.705382, 0.049364], [0,0,0,0], [9E9, 9E9, 9E9, 9E9, 9E9, 9E9]];
	VAR robtarget OpenholeUD_5940 := [[449.05, -29.1, 181.71], [0.034567, 0.706261, 0.706193, 0.035944], [0,0,0,0], [9E9, 9E9, 9E9, 9E9, 9E9, 9E9]];
	VAR robtarget OpenholeUD_5941 := [[453.03, -29.1, 182.1], [0.048119, 0.705468, 0.70675, 0.022455], [0,0,0,0], [9E9, 9E9, 9E9, 9E9, 9E9, 9E9]];
	VAR robtarget OpenholeUD_5942 := [[457.01, -29.1, 182.48], [0.061562, 0.704422, 0.70705, 0.00894], [0,0,0,0], [9E9, 9E9, 9E9, 9E9, 9E9, 9E9]];
	VAR robtarget OpenholeUD_5943 := [[460.99, -29.1, 182.87], [0.074851, 0.703134, 0.707092, -0.004555], [0,0,0,0], [9E9, 9E9, 9E9, 9E9, 9E9, 9E9]];
	VAR robtarget OpenholeUD_5944 := [[464.97, -29.1, 183.26], [0.087946, 0.701616, 0.706878, -0.017988], [0,0,0,0], [9E9, 9E9, 9E9, 9E9, 9E9, 9E9]];
	VAR robtarget OpenholeUD_5945 := [[468.96, -29.1, 183.64], [0.100811, 0.699884, 0.706413, -0.031316], [0,0,0,0], [9E9, 9E9, 9E9, 9E9, 9E9, 9E9]];
	VAR robtarget OpenholeUD_5946 := [[472.94, -29.1, 184.03], [0.113412, 0.697953, 0.705705, -0.0445], [0,0,0,0], [9E9, 9E9, 9E9, 9E9, 9E9, 9E9]];
	VAR robtarget OpenholeUD_5947 := [[476.92, -29.1, 184.41], [0.125721, 0.695841, 0.704765, -0.057501], [0,0,0,0], [9E9, 9E9, 9E9, 9E9, 9E9, 9E9]];
	VAR robtarget OpenholeUD_5948 := [[480.9, -29.1, 184.8], [0.137712, 0.693567, 0.703605, -0.070286], [0,0,0,0], [9E9, 9E9, 9E9, 9E9, 9E9, 9E9]];
	VAR robtarget OpenholeUD_5949 := [[484.88, -29.1, 185.19], [0.149365, 0.691151, 0.702239, -0.082825], [0,0,0,0], [9E9, 9E9, 9E9, 9E9, 9E9, 9E9]];
	VAR robtarget OpenholeUD_5950 := [[488.86, -29.1, 185.57], [0.160664, 0.688612, 0.700684, -0.09509], [0,0,0,0], [9E9, 9E9, 9E9, 9E9, 9E9, 9E9]];
	VAR robtarget OpenholeUD_5951 := [[492.84, -29.1, 185.96], [0.171599, 0.685969, 0.698955, -0.10706], [0,0,0,0], [9E9, 9E9, 9E9, 9E9, 9E9, 9E9]];
	VAR robtarget OpenholeUD_5952 := [[496.83, -29.1, 186.34], [0.18216, 0.683241, 0.69707, -0.118715], [0,0,0,0], [9E9, 9E9, 9E9, 9E9, 9E9, 9E9]];
	VAR robtarget OpenholeUD_5953 := [[500.81, -29.1, 186.73], [0.192343, 0.680444, 0.695046, -0.13004], [0,0,0,0], [9E9, 9E9, 9E9, 9E9, 9E9, 9E9]];
	VAR robtarget OpenholeUD_5954 := [[504.79, -29.1, 187.12], [0.202149, 0.677596, 0.692901, -0.141026], [0,0,0,0], [9E9, 9E9, 9E9, 9E9, 9E9, 9E9]];
	VAR robtarget OpenholeUD_5955 := [[509.37, -29.1, 187.56], [0.183051, 0.683002, 0.683002, -0.183051], [0,0,0,0], [9E9, 9E9, 9E9, 9E9, 9E9, 9E9]];
	VAR robtarget OpenholeUD_5956 := [[513.37, -29.1, 187.55], [0.183051, 0.683002, 0.683002, -0.183051], [0,0,0,0], [9E9, 9E9, 9E9, 9E9, 9E9, 9E9]];
	VAR robtarget OpenholeUD_5957 := [[517.37, -29.1, 187.53], [0.183051, 0.683002, 0.683002, -0.183051], [0,0,0,0], [9E9, 9E9, 9E9, 9E9, 9E9, 9E9]];
	VAR robtarget OpenholeUD_5958 := [[521.37, -29.1, 187.52], [0.183051, 0.683002, 0.683002, -0.183051], [0,0,0,0], [9E9, 9E9, 9E9, 9E9, 9E9, 9E9]];
	VAR robtarget OpenholeUD_5959 := [[525.37, -29.1, 187.51], [0.183051, 0.683002, 0.683002, -0.183051], [0,0,0,0], [9E9, 9E9, 9E9, 9E9, 9E9, 9E9]];
	VAR robtarget OpenholeUD_5960 := [[529.37, -29.1, 187.5], [0.183051, 0.683002, 0.683002, -0.183051], [0,0,0,0], [9E9, 9E9, 9E9, 9E9, 9E9, 9E9]];
	VAR robtarget OpenholeUD_5961 := [[529.37, -29.1, 187.5], [0.183051, 0.683002, 0.683002, -0.183051], [0,0,0,0], [9E9, 9E9, 9E9, 9E9, 9E9, 9E9]];
	VAR robtarget OpenholeUD_5962 := [[529.36, -27.9, 186.8], [0.183051, 0.683002, 0.683002, -0.183051], [0,0,0,0], [9E9, 9E9, 9E9, 9E9, 9E9, 9E9]];
	VAR robtarget OpenholeUD_5963 := [[525.36, -27.9, 186.82], [0.183051, 0.683002, 0.683002, -0.183051], [0,0,0,0], [9E9, 9E9, 9E9, 9E9, 9E9, 9E9]];
	VAR robtarget OpenholeUD_5964 := [[521.36, -27.9, 186.83], [0.183051, 0.683002, 0.683002, -0.183051], [0,0,0,0], [9E9, 9E9, 9E9, 9E9, 9E9, 9E9]];
	VAR robtarget OpenholeUD_5965 := [[517.36, -27.9, 186.84], [0.183051, 0.683002, 0.683002, -0.183051], [0,0,0,0], [9E9, 9E9, 9E9, 9E9, 9E9, 9E9]];
	VAR robtarget OpenholeUD_5966 := [[513.36, -27.9, 186.85], [0.183051, 0.683002, 0.683002, -0.183051], [0,0,0,0], [9E9, 9E9, 9E9, 9E9, 9E9, 9E9]];
	VAR robtarget OpenholeUD_5967 := [[509.36, -27.9, 186.87], [0.183051, 0.683002, 0.683002, -0.183051], [0,0,0,0], [9E9, 9E9, 9E9, 9E9, 9E9, 9E9]];
	VAR robtarget OpenholeUD_5968 := [[505.38, -27.9, 186.53], [0.200147, 0.67819, 0.691847, -0.14611], [0,0,0,0], [9E9, 9E9, 9E9, 9E9, 9E9, 9E9]];
	VAR robtarget OpenholeUD_5969 := [[501.39, -27.9, 186.19], [0.190319, 0.681013, 0.694056, -0.135229], [0,0,0,0], [9E9, 9E9, 9E9, 9E9, 9E9, 9E9]];
	VAR robtarget OpenholeUD_5970 := [[497.41, -27.9, 185.85], [0.180113, 0.683783, 0.696149, -0.124004], [0,0,0,0], [9E9, 9E9, 9E9, 9E9, 9E9, 9E9]];
	VAR robtarget OpenholeUD_5971 := [[493.42, -27.9, 185.5], [0.16953, 0.686483, 0.698109, -0.112444], [0,0,0,0], [9E9, 9E9, 9E9, 9E9, 9E9, 9E9]];
	VAR robtarget OpenholeUD_5972 := [[489.44, -27.9, 185.16], [0.158575, 0.689096, 0.699919, -0.100564], [0,0,0,0], [9E9, 9E9, 9E9, 9E9, 9E9, 9E9]];
	VAR robtarget OpenholeUD_5973 := [[485.45, -27.9, 184.82], [0.147256, 0.691604, 0.701562, -0.088381], [0,0,0,0], [9E9, 9E9, 9E9, 9E9, 9E9, 9E9]];
	VAR robtarget OpenholeUD_5974 := [[481.47, -27.9, 184.48], [0.135583, 0.693986, 0.70302, -0.075917], [0,0,0,0], [9E9, 9E9, 9E9, 9E9, 9E9, 9E9]];
	VAR robtarget OpenholeUD_5975 := [[477.48, -27.9, 184.14], [0.123574, 0.696225, 0.704277, -0.063196], [0,0,0,0], [9E9, 9E9, 9E9, 9E9, 9E9, 9E9]];
	VAR robtarget OpenholeUD_5976 := [[473.49, -27.9, 183.8], [0.111249, 0.698301, 0.705319, -0.05025], [0,0,0,0], [9E9, 9E9, 9E9, 9E9, 9E9, 9E9]];
	VAR robtarget OpenholeUD_5977 := [[469.51, -27.9, 183.46], [0.098632, 0.700194, 0.706132, -0.03711], [0,0,0,0], [9E9, 9E9, 9E9, 9E9, 9E9, 9E9]];
	VAR robtarget OpenholeUD_5978 := [[465.52, -27.9, 183.12], [0.085752, 0.701888, 0.706706, -0.023813], [0,0,0,0], [9E9, 9E9, 9E9, 9E9, 9E9, 9E9]];
	VAR robtarget OpenholeUD_5979 := [[461.54, -27.9, 182.78], [0.072642, 0.703366, 0.70703, -0.0104], [0,0,0,0], [9E9, 9E9, 9E9, 9E9, 9E9, 9E9]];
	VAR robtarget OpenholeUD_5980 := [[457.55, -27.9, 182.44], [0.05934, 0.704612, 0.7071, 0.003089], [0,0,0,0], [9E9, 9E9, 9E9, 9E9, 9E9, 9E9]];
	VAR robtarget OpenholeUD_5981 := [[453.57, -27.9, 182.1], [0.045886, 0.705616, 0.706912, 0.01661], [0,0,0,0], [9E9, 9E9, 9E9, 9E9, 9E9, 9E9]];
	VAR robtarget OpenholeUD_5982 := [[449.58, -27.9, 181.76], [0.032323, 0.706368, 0.706465, 0.030118], [0,0,0,0], [9E9, 9E9, 9E9, 9E9, 9E9, 9E9]];
	VAR robtarget OpenholeUD_5983 := [[445.6, -27.9, 181.42], [0.018695, 0.70686, 0.705763, 0.043571], [0,0,0,0], [9E9, 9E9, 9E9, 9E9, 9E9, 9E9]];
	VAR robtarget OpenholeUD_5984 := [[441.61, -27.9, 181.08], [0.005048, 0.707089, 0.704812, 0.056924], [0,0,0,0], [9E9, 9E9, 9E9, 9E9, 9E9, 9E9]];
	VAR robtarget OpenholeUD_5985 := [[437.62, -27.9, 180.74], [-0.008572, 0.707055, 0.70362, 0.070136], [0,0,0,0], [9E9, 9E9, 9E9, 9E9, 9E9, 9E9]];
	VAR robtarget OpenholeUD_5986 := [[433.64, -27.9, 180.4], [-0.022119, 0.706761, 0.702199, 0.083168], [0,0,0,0], [9E9, 9E9, 9E9, 9E9, 9E9, 9E9]];
	VAR robtarget OpenholeUD_5987 := [[429.65, -27.9, 180.06], [-0.03555, 0.706213, 0.700562, 0.095983], [0,0,0,0], [9E9, 9E9, 9E9, 9E9, 9E9, 9E9]];
	VAR robtarget OpenholeUD_5988 := [[425.67, -27.9, 179.72], [-0.048825, 0.705419, 0.698725, 0.108549], [0,0,0,0], [9E9, 9E9, 9E9, 9E9, 9E9, 9E9]];
	VAR robtarget OpenholeUD_5989 := [[421.68, -27.9, 179.38], [-0.061904, 0.704392, 0.696706, 0.120836], [0,0,0,0], [9E9, 9E9, 9E9, 9E9, 9E9, 9E9]];
	VAR robtarget OpenholeUD_5990 := [[417.7, -27.9, 179.04], [-0.074753, 0.703144, 0.694521, 0.13282], [0,0,0,0], [9E9, 9E9, 9E9, 9E9, 9E9, 9E9]];
	VAR robtarget OpenholeUD_5991 := [[413.71, -27.9, 178.7], [-0.087342, 0.701692, 0.692189, 0.144479], [0,0,0,0], [9E9, 9E9, 9E9, 9E9, 9E9, 9E9]];
	VAR robtarget OpenholeUD_5992 := [[409.73, -27.9, 178.36], [-0.099643, 0.700051, 0.68973, 0.155798], [0,0,0,0], [9E9, 9E9, 9E9, 9E9, 9E9, 9E9]];
	VAR robtarget OpenholeUD_5993 := [[405.74, -27.9, 178.02], [-0.111635, 0.698239, 0.687161, 0.166763], [0,0,0,0], [9E9, 9E9, 9E9, 9E9, 9E9, 9E9]];
	VAR robtarget OpenholeUD_5994 := [[401.76, -27.9, 177.68], [-0.123299, 0.696274, 0.684501, 0.177367], [0,0,0,0], [9E9, 9E9, 9E9, 9E9, 9E9, 9E9]];
	VAR robtarget OpenholeUD_5995 := [[397.77, -27.9, 177.34], [-0.134622, 0.694174, 0.681766, 0.187602], [0,0,0,0], [9E9, 9E9, 9E9, 9E9, 9E9, 9E9]];
	VAR robtarget OpenholeUD_5996 := [[393.78, -27.9, 177], [-0.145593, 0.691956, 0.678974, 0.197468], [0,0,0,0], [9E9, 9E9, 9E9, 9E9, 9E9, 9E9]];
	VAR robtarget OpenholeUD_5997 := [[389.33, -27.9, 176.62], [-0.157427, 0.68936, 0.675805, 0.208057], [0,0,0,0], [9E9, 9E9, 9E9, 9E9, 9E9, 9E9]];
	VAR robtarget OpenholeUD_5998 := [[385.33, -27.9, 176.63], [-0.183051, 0.683002, 0.683002, 0.183051], [0,0,0,0], [9E9, 9E9, 9E9, 9E9, 9E9, 9E9]];
	VAR robtarget OpenholeUD_5999 := [[381.33, -27.9, 176.64], [-0.183051, 0.683002, 0.683002, 0.183051], [0,0,0,0], [9E9, 9E9, 9E9, 9E9, 9E9, 9E9]];
	VAR robtarget OpenholeUD_6000 := [[377.33, -27.9, 176.65], [-0.183051, 0.683002, 0.683002, 0.183051], [0,0,0,0], [9E9, 9E9, 9E9, 9E9, 9E9, 9E9]];
	VAR robtarget OpenholeUD_6001 := [[373.33, -27.9, 176.67], [-0.183051, 0.683002, 0.683002, 0.183051], [0,0,0,0], [9E9, 9E9, 9E9, 9E9, 9E9, 9E9]];
	VAR robtarget OpenholeUD_6002 := [[369.33, -27.9, 176.68], [-0.183051, 0.683002, 0.683002, 0.183051], [0,0,0,0], [9E9, 9E9, 9E9, 9E9, 9E9, 9E9]];
	VAR robtarget OpenholeUD_6003 := [[369.33, -27.9, 176.68], [-0.183051, 0.683002, 0.683002, 0.183051], [0,0,0,0], [9E9, 9E9, 9E9, 9E9, 9E9, 9E9]];
	VAR robtarget OpenholeUD_6004 := [[369.33, -26.7, 177.37], [-0.183051, 0.683002, 0.683002, 0.183051], [0,0,0,0], [9E9, 9E9, 9E9, 9E9, 9E9, 9E9]];
	VAR robtarget OpenholeUD_6005 := [[373.33, -26.7, 177.36], [-0.183051, 0.683002, 0.683002, 0.183051], [0,0,0,0], [9E9, 9E9, 9E9, 9E9, 9E9, 9E9]];
	VAR robtarget OpenholeUD_6006 := [[377.33, -26.7, 177.35], [-0.183051, 0.683002, 0.683002, 0.183051], [0,0,0,0], [9E9, 9E9, 9E9, 9E9, 9E9, 9E9]];
	VAR robtarget OpenholeUD_6007 := [[381.33, -26.7, 177.34], [-0.183051, 0.683002, 0.683002, 0.183051], [0,0,0,0], [9E9, 9E9, 9E9, 9E9, 9E9, 9E9]];
	VAR robtarget OpenholeUD_6008 := [[385.33, -26.7, 177.32], [-0.183051, 0.683002, 0.683002, 0.183051], [0,0,0,0], [9E9, 9E9, 9E9, 9E9, 9E9, 9E9]];
	VAR robtarget OpenholeUD_6009 := [[389.33, -26.7, 177.31], [-0.160868, 0.688565, 0.67683, 0.204696], [0,0,0,0], [9E9, 9E9, 9E9, 9E9, 9E9, 9E9]];
	VAR robtarget OpenholeUD_6010 := [[393.32, -26.7, 177.6], [-0.150356, 0.690936, 0.67964, 0.195165], [0,0,0,0], [9E9, 9E9, 9E9, 9E9, 9E9, 9E9]];
	VAR robtarget OpenholeUD_6011 := [[397.31, -26.7, 177.9], [-0.139484, 0.693213, 0.682405, 0.185265], [0,0,0,0], [9E9, 9E9, 9E9, 9E9, 9E9, 9E9]];
	VAR robtarget OpenholeUD_6012 := [[401.3, -26.7, 178.19], [-0.128256, 0.695378, 0.68511, 0.174996], [0,0,0,0], [9E9, 9E9, 9E9, 9E9, 9E9, 9E9]];
	VAR robtarget OpenholeUD_6013 := [[405.29, -26.7, 178.49], [-0.116682, 0.697413, 0.687739, 0.164361], [0,0,0,0], [9E9, 9E9, 9E9, 9E9, 9E9, 9E9]];
	VAR robtarget OpenholeUD_6014 := [[409.28, -26.7, 178.78], [-0.104774, 0.699301, 0.690275, 0.153365], [0,0,0,0], [9E9, 9E9, 9E9, 9E9, 9E9, 9E9]];
	VAR robtarget OpenholeUD_6015 := [[413.27, -26.7, 179.08], [-0.092551, 0.701024, 0.692698, 0.142017], [0,0,0,0], [9E9, 9E9, 9E9, 9E9, 9E9, 9E9]];
	VAR robtarget OpenholeUD_6016 := [[417.26, -26.7, 179.37], [-0.080033, 0.702563, 0.694992, 0.13033], [0,0,0,0], [9E9, 9E9, 9E9, 9E9, 9E9, 9E9]];
	VAR robtarget OpenholeUD_6017 := [[421.25, -26.7, 179.67], [-0.067246, 0.703902, 0.697137, 0.11832], [0,0,0,0], [9E9, 9E9, 9E9, 9E9, 9E9, 9E9]];
	VAR robtarget OpenholeUD_6018 := [[425.24, -26.7, 179.96], [-0.054219, 0.705025, 0.699115, 0.106008], [0,0,0,0], [9E9, 9E9, 9E9, 9E9, 9E9, 9E9]];
	VAR robtarget OpenholeUD_6019 := [[429.22, -26.7, 180.26], [-0.040987, 0.705918, 0.700909, 0.093419], [0,0,0,0], [9E9, 9E9, 9E9, 9E9, 9E9, 9E9]];
	VAR robtarget OpenholeUD_6020 := [[433.21, -26.7, 180.55], [-0.027587, 0.706568, 0.7025, 0.080584], [0,0,0,0], [9E9, 9E9, 9E9, 9E9, 9E9, 9E9]];
	VAR robtarget OpenholeUD_6021 := [[437.2, -26.7, 180.84], [-0.014059, 0.706967, 0.703874, 0.067534], [0,0,0,0], [9E9, 9E9, 9E9, 9E9, 9E9, 9E9]];
	VAR robtarget OpenholeUD_6022 := [[441.19, -26.7, 181.14], [-0.000447, 0.707107, 0.705018, 0.054306], [0,0,0,0], [9E9, 9E9, 9E9, 9E9, 9E9, 9E9]];
	VAR robtarget OpenholeUD_6023 := [[445.18, -26.7, 181.43], [0.013204, 0.706983, 0.705921, 0.040939], [0,0,0,0], [9E9, 9E9, 9E9, 9E9, 9E9, 9E9]];
	VAR robtarget OpenholeUD_6024 := [[449.17, -26.7, 181.73], [0.026848, 0.706597, 0.706573, 0.027475], [0,0,0,0], [9E9, 9E9, 9E9, 9E9, 9E9, 9E9]];
	VAR robtarget OpenholeUD_6025 := [[453.16, -26.7, 182.02], [0.04044, 0.705949, 0.706969, 0.013958], [0,0,0,0], [9E9, 9E9, 9E9, 9E9, 9E9, 9E9]];
	VAR robtarget OpenholeUD_6026 := [[457.15, -26.7, 182.32], [0.053935, 0.705047, 0.707107, 0.000432], [0,0,0,0], [9E9, 9E9, 9E9, 9E9, 9E9, 9E9]];
	VAR robtarget OpenholeUD_6027 := [[461.14, -26.7, 182.61], [0.067289, 0.703898, 0.706986, -0.01306], [0,0,0,0], [9E9, 9E9, 9E9, 9E9, 9E9, 9E9]];
	VAR robtarget OpenholeUD_6028 := [[465.13, -26.7, 182.91], [0.08046, 0.702514, 0.706611, -0.026474], [0,0,0,0], [9E9, 9E9, 9E9, 9E9, 9E9, 9E9]];
	VAR robtarget OpenholeUD_6029 := [[469.12, -26.7, 183.2], [0.093412, 0.70091, 0.705988, -0.039768], [0,0,0,0], [9E9, 9E9, 9E9, 9E9, 9E9, 9E9]];
	VAR robtarget OpenholeUD_6030 := [[473.11, -26.7, 183.5], [0.106109, 0.6991, 0.705125, -0.052903], [0,0,0,0], [9E9, 9E9, 9E9, 9E9, 9E9, 9E9]];
	VAR robtarget OpenholeUD_6031 := [[477.09, -26.7, 183.79], [0.118522, 0.697103, 0.704035, -0.065842], [0,0,0,0], [9E9, 9E9, 9E9, 9E9, 9E9, 9E9]];
	VAR robtarget OpenholeUD_6032 := [[481.08, -26.7, 184.08], [0.130625, 0.694937, 0.70273, -0.078552], [0,0,0,0], [9E9, 9E9, 9E9, 9E9, 9E9, 9E9]];
	VAR robtarget OpenholeUD_6033 := [[485.07, -26.7, 184.38], [0.142397, 0.69262, 0.701226, -0.091003], [0,0,0,0], [9E9, 9E9, 9E9, 9E9, 9E9, 9E9]];
	VAR robtarget OpenholeUD_6034 := [[489.06, -26.7, 184.67], [0.153821, 0.690173, 0.69954, -0.103171], [0,0,0,0], [9E9, 9E9, 9E9, 9E9, 9E9, 9E9]];
	VAR robtarget OpenholeUD_6035 := [[493.05, -26.7, 184.97], [0.164883, 0.687614, 0.697687, -0.115033], [0,0,0,0], [9E9, 9E9, 9E9, 9E9, 9E9, 9E9]];
	VAR robtarget OpenholeUD_6036 := [[497.04, -26.7, 185.26], [0.175575, 0.684962, 0.695686, -0.126573], [0,0,0,0], [9E9, 9E9, 9E9, 9E9, 9E9, 9E9]];
	VAR robtarget OpenholeUD_6037 := [[501.03, -26.7, 185.56], [0.185893, 0.682234, 0.693554, -0.137776], [0,0,0,0], [9E9, 9E9, 9E9, 9E9, 9E9, 9E9]];
	VAR robtarget OpenholeUD_6038 := [[505.02, -26.7, 185.85], [0.195833, 0.679448, 0.691309, -0.148633], [0,0,0,0], [9E9, 9E9, 9E9, 9E9, 9E9, 9E9]];
	VAR robtarget OpenholeUD_6039 := [[509.36, -26.7, 186.17], [0.183051, 0.683002, 0.683002, -0.183051], [0,0,0,0], [9E9, 9E9, 9E9, 9E9, 9E9, 9E9]];
	VAR robtarget OpenholeUD_6040 := [[513.36, -26.7, 186.16], [0.183051, 0.683002, 0.683002, -0.183051], [0,0,0,0], [9E9, 9E9, 9E9, 9E9, 9E9, 9E9]];
	VAR robtarget OpenholeUD_6041 := [[517.36, -26.7, 186.15], [0.183051, 0.683002, 0.683002, -0.183051], [0,0,0,0], [9E9, 9E9, 9E9, 9E9, 9E9, 9E9]];
	VAR robtarget OpenholeUD_6042 := [[521.36, -26.7, 186.14], [0.183051, 0.683002, 0.683002, -0.183051], [0,0,0,0], [9E9, 9E9, 9E9, 9E9, 9E9, 9E9]];
	VAR robtarget OpenholeUD_6043 := [[525.36, -26.7, 186.12], [0.183051, 0.683002, 0.683002, -0.183051], [0,0,0,0], [9E9, 9E9, 9E9, 9E9, 9E9, 9E9]];
	VAR robtarget OpenholeUD_6044 := [[529.36, -26.7, 186.11], [0.183051, 0.683002, 0.683002, -0.183051], [0,0,0,0], [9E9, 9E9, 9E9, 9E9, 9E9, 9E9]];
	VAR robtarget OpenholeUD_6045 := [[529.36, -26.7, 186.11], [0.183051, 0.683002, 0.683002, -0.183051], [0,0,0,0], [9E9, 9E9, 9E9, 9E9, 9E9, 9E9]];
	VAR robtarget OpenholeUD_6046 := [[529.36, -25.5, 185.42], [0.183051, 0.683002, 0.683002, -0.183051], [0,0,0,0], [9E9, 9E9, 9E9, 9E9, 9E9, 9E9]];
	VAR robtarget OpenholeUD_6047 := [[525.36, -25.5, 185.43], [0.183051, 0.683002, 0.683002, -0.183051], [0,0,0,0], [9E9, 9E9, 9E9, 9E9, 9E9, 9E9]];
	VAR robtarget OpenholeUD_6048 := [[521.36, -25.5, 185.44], [0.183051, 0.683002, 0.683002, -0.183051], [0,0,0,0], [9E9, 9E9, 9E9, 9E9, 9E9, 9E9]];
	VAR robtarget OpenholeUD_6049 := [[517.36, -25.5, 185.45], [0.183051, 0.683002, 0.683002, -0.183051], [0,0,0,0], [9E9, 9E9, 9E9, 9E9, 9E9, 9E9]];
	VAR robtarget OpenholeUD_6050 := [[513.36, -25.5, 185.47], [0.183051, 0.683002, 0.683002, -0.183051], [0,0,0,0], [9E9, 9E9, 9E9, 9E9, 9E9, 9E9]];
	VAR robtarget OpenholeUD_6051 := [[509.36, -25.5, 185.48], [0.183051, 0.683002, 0.683002, -0.183051], [0,0,0,0], [9E9, 9E9, 9E9, 9E9, 9E9, 9E9]];
	VAR robtarget OpenholeUD_6052 := [[505.37, -25.5, 185.23], [0.19324, 0.68019, 0.690344, -0.153053], [0,0,0,0], [9E9, 9E9, 9E9, 9E9, 9E9, 9E9]];
	VAR robtarget OpenholeUD_6053 := [[501.38, -25.5, 184.98], [0.183255, 0.682948, 0.692644, -0.142284], [0,0,0,0], [9E9, 9E9, 9E9, 9E9, 9E9, 9E9]];
	VAR robtarget OpenholeUD_6054 := [[497.38, -25.5, 184.73], [0.172895, 0.685644, 0.694835, -0.131166], [0,0,0,0], [9E9, 9E9, 9E9, 9E9, 9E9, 9E9]];
	VAR robtarget OpenholeUD_6055 := [[493.39, -25.5, 184.49], [0.16216, 0.688262, 0.6969, -0.119707], [0,0,0,0], [9E9, 9E9, 9E9, 9E9, 9E9, 9E9]];
	VAR robtarget OpenholeUD_6056 := [[489.4, -25.5, 184.24], [0.151057, 0.690783, 0.698823, -0.107921], [0,0,0,0], [9E9, 9E9, 9E9, 9E9, 9E9, 9E9]];
	VAR robtarget OpenholeUD_6057 := [[485.41, -25.5, 183.99], [0.139594, 0.693191, 0.700584, -0.095823], [0,0,0,0], [9E9, 9E9, 9E9, 9E9, 9E9, 9E9]];
	VAR robtarget OpenholeUD_6058 := [[481.41, -25.5, 183.74], [0.127785, 0.695465, 0.702167, -0.083436], [0,0,0,0], [9E9, 9E9, 9E9, 9E9, 9E9, 9E9]];
	VAR robtarget OpenholeUD_6059 := [[477.42, -25.5, 183.49], [0.115647, 0.697586, 0.703555, -0.070782], [0,0,0,0], [9E9, 9E9, 9E9, 9E9, 9E9, 9E9]];
	VAR robtarget OpenholeUD_6060 := [[473.43, -25.5, 183.24], [0.103201, 0.699535, 0.704733, -0.057891], [0,0,0,0], [9E9, 9E9, 9E9, 9E9, 9E9, 9E9]];
	VAR robtarget OpenholeUD_6061 := [[469.44, -25.5, 182.99], [0.090474, 0.701295, 0.705686, -0.044796], [0,0,0,0], [9E9, 9E9, 9E9, 9E9, 9E9, 9E9]];
	VAR robtarget OpenholeUD_6062 := [[465.44, -25.5, 182.74], [0.077496, 0.702847, 0.706403, -0.031532], [0,0,0,0], [9E9, 9E9, 9E9, 9E9, 9E9, 9E9]];
	VAR robtarget OpenholeUD_6063 := [[461.45, -25.5, 182.5], [0.064301, 0.704177, 0.706874, -0.018138], [0,0,0,0], [9E9, 9E9, 9E9, 9E9, 9E9, 9E9]];
	VAR robtarget OpenholeUD_6064 := [[457.46, -25.5, 182.25], [0.050927, 0.70527, 0.707091, -0.004656], [0,0,0,0], [9E9, 9E9, 9E9, 9E9, 9E9, 9E9]];
	VAR robtarget OpenholeUD_6065 := [[453.47, -25.5, 182], [0.037417, 0.706116, 0.707051, 0.008872], [0,0,0,0], [9E9, 9E9, 9E9, 9E9, 9E9, 9E9]];
	VAR robtarget OpenholeUD_6066 := [[449.48, -25.5, 181.75], [0.023812, 0.706706, 0.706752, 0.022401], [0,0,0,0], [9E9, 9E9, 9E9, 9E9, 9E9, 9E9]];
	VAR robtarget OpenholeUD_6067 := [[445.48, -25.5, 181.5], [0.010159, 0.707034, 0.706196, 0.035886], [0,0,0,0], [9E9, 9E9, 9E9, 9E9, 9E9, 9E9]];
	VAR robtarget OpenholeUD_6068 := [[441.49, -25.5, 181.25], [-0.003497, 0.707098, 0.705387, 0.049286], [0,0,0,0], [9E9, 9E9, 9E9, 9E9, 9E9, 9E9]];
	VAR robtarget OpenholeUD_6069 := [[437.5, -25.5, 181], [-0.017109, 0.7069, 0.704334, 0.062556], [0,0,0,0], [9E9, 9E9, 9E9, 9E9, 9E9, 9E9]];
	VAR robtarget OpenholeUD_6070 := [[433.51, -25.5, 180.75], [-0.030633, 0.706443, 0.703048, 0.075658], [0,0,0,0], [9E9, 9E9, 9E9, 9E9, 9E9, 9E9]];
	VAR robtarget OpenholeUD_6071 := [[429.51, -25.5, 180.51], [-0.044026, 0.705735, 0.70154, 0.088554], [0,0,0,0], [9E9, 9E9, 9E9, 9E9, 9E9, 9E9]];
	VAR robtarget OpenholeUD_6072 := [[425.52, -25.5, 180.26], [-0.057246, 0.704786, 0.699826, 0.101211], [0,0,0,0], [9E9, 9E9, 9E9, 9E9, 9E9, 9E9]];
	VAR robtarget OpenholeUD_6073 := [[421.53, -25.5, 180.01], [-0.070258, 0.703608, 0.697922, 0.113597], [0,0,0,0], [9E9, 9E9, 9E9, 9E9, 9E9, 9E9]];
	VAR robtarget OpenholeUD_6074 := [[417.54, -25.5, 179.76], [-0.083026, 0.702216, 0.695846, 0.125689], [0,0,0,0], [9E9, 9E9, 9E9, 9E9, 9E9, 9E9]];
	VAR robtarget OpenholeUD_6075 := [[413.55, -25.5, 179.51], [-0.095522, 0.700625, 0.693617, 0.137463], [0,0,0,0], [9E9, 9E9, 9E9, 9E9, 9E9, 9E9]];
	VAR robtarget OpenholeUD_6076 := [[409.55, -25.5, 179.26], [-0.10772, 0.698854, 0.691251, 0.148902], [0,0,0,0], [9E9, 9E9, 9E9, 9E9, 9E9, 9E9]];
	VAR robtarget OpenholeUD_6077 := [[405.56, -25.5, 179.01], [-0.119599, 0.696919, 0.688769, 0.159992], [0,0,0,0], [9E9, 9E9, 9E9, 9E9, 9E9, 9E9]];
	VAR robtarget OpenholeUD_6078 := [[401.57, -25.5, 178.77], [-0.131142, 0.694839, 0.686188, 0.170724], [0,0,0,0], [9E9, 9E9, 9E9, 9E9, 9E9, 9E9]];
	VAR robtarget OpenholeUD_6079 := [[397.58, -25.5, 178.52], [-0.142337, 0.692633, 0.683525, 0.181091], [0,0,0,0], [9E9, 9E9, 9E9, 9E9, 9E9, 9E9]];
	VAR robtarget OpenholeUD_6080 := [[393.58, -25.5, 178.27], [-0.153174, 0.690317, 0.680797, 0.19109], [0,0,0,0], [9E9, 9E9, 9E9, 9E9, 9E9, 9E9]];
	VAR robtarget OpenholeUD_6081 := [[389.34, -25.5, 178], [-0.164309, 0.687752, 0.67784, 0.201327], [0,0,0,0], [9E9, 9E9, 9E9, 9E9, 9E9, 9E9]];
	VAR robtarget OpenholeUD_6082 := [[385.34, -25.5, 178.02], [-0.183051, 0.683002, 0.683002, 0.183051], [0,0,0,0], [9E9, 9E9, 9E9, 9E9, 9E9, 9E9]];
	VAR robtarget OpenholeUD_6083 := [[381.34, -25.5, 178.03], [-0.183051, 0.683002, 0.683002, 0.183051], [0,0,0,0], [9E9, 9E9, 9E9, 9E9, 9E9, 9E9]];
	VAR robtarget OpenholeUD_6084 := [[377.34, -25.5, 178.04], [-0.183051, 0.683002, 0.683002, 0.183051], [0,0,0,0], [9E9, 9E9, 9E9, 9E9, 9E9, 9E9]];
	VAR robtarget OpenholeUD_6085 := [[373.34, -25.5, 178.05], [-0.183051, 0.683002, 0.683002, 0.183051], [0,0,0,0], [9E9, 9E9, 9E9, 9E9, 9E9, 9E9]];
	VAR robtarget OpenholeUD_6086 := [[369.34, -25.5, 178.07], [-0.183051, 0.683002, 0.683002, 0.183051], [0,0,0,0], [9E9, 9E9, 9E9, 9E9, 9E9, 9E9]];
	VAR robtarget OpenholeUD_6087 := [[369.34, -25.5, 178.07], [-0.183051, 0.683002, 0.683002, 0.183051], [0,0,0,0], [9E9, 9E9, 9E9, 9E9, 9E9, 9E9]];
	VAR robtarget OpenholeUD_6088 := [[369.34, -24.3, 178.76], [-0.183051, 0.683002, 0.683002, 0.183051], [0,0,0,0], [9E9, 9E9, 9E9, 9E9, 9E9, 9E9]];
	VAR robtarget OpenholeUD_6089 := [[373.34, -24.3, 178.75], [-0.183051, 0.683002, 0.683002, 0.183051], [0,0,0,0], [9E9, 9E9, 9E9, 9E9, 9E9, 9E9]];
	VAR robtarget OpenholeUD_6090 := [[377.34, -24.3, 178.73], [-0.183051, 0.683002, 0.683002, 0.183051], [0,0,0,0], [9E9, 9E9, 9E9, 9E9, 9E9, 9E9]];
	VAR robtarget OpenholeUD_6091 := [[381.34, -24.3, 178.72], [-0.183051, 0.683002, 0.683002, 0.183051], [0,0,0,0], [9E9, 9E9, 9E9, 9E9, 9E9, 9E9]];
	VAR robtarget OpenholeUD_6092 := [[389.34, -24.3, 178.7], [-0.167749, 0.686921, 0.678834, 0.19795], [0,0,0,0], [9E9, 9E9, 9E9, 9E9, 9E9, 9E9]];
	VAR robtarget OpenholeUD_6093 := [[393.33, -24.3, 178.9], [-0.15736, 0.689375, 0.681583, 0.188266], [0,0,0,0], [9E9, 9E9, 9E9, 9E9, 9E9, 9E9]];
	VAR robtarget OpenholeUD_6094 := [[397.33, -24.3, 179.1], [-0.146606, 0.691742, 0.68428, 0.178216], [0,0,0,0], [9E9, 9E9, 9E9, 9E9, 9E9, 9E9]];
	VAR robtarget OpenholeUD_6095 := [[401.32, -24.3, 179.3], [-0.135492, 0.694004, 0.686909, 0.167799], [0,0,0,0], [9E9, 9E9, 9E9, 9E9, 9E9, 9E9]];
	VAR robtarget OpenholeUD_6096 := [[405.32, -24.3, 179.51], [-0.124026, 0.696145, 0.689453, 0.157018], [0,0,0,0], [9E9, 9E9, 9E9, 9E9, 9E9, 9E9]];
	VAR robtarget OpenholeUD_6097 := [[409.31, -24.3, 179.71], [-0.11222, 0.698145, 0.691895, 0.145881], [0,0,0,0], [9E9, 9E9, 9E9, 9E9, 9E9, 9E9]];
	VAR robtarget OpenholeUD_6098 := [[413.31, -24.3, 179.91], [-0.100089, 0.699987, 0.694217, 0.134397], [0,0,0,0], [9E9, 9E9, 9E9, 9E9, 9E9, 9E9]];
	VAR robtarget OpenholeUD_6099 := [[417.3, -24.3, 180.12], [-0.087655, 0.701653, 0.696401, 0.122581], [0,0,0,0], [9E9, 9E9, 9E9, 9E9, 9E9, 9E9]];
	VAR robtarget OpenholeUD_6100 := [[421.3, -24.3, 180.32], [-0.074941, 0.703124, 0.698427, 0.11045], [0,0,0,0], [9E9, 9E9, 9E9, 9E9, 9E9, 9E9]];
	VAR robtarget OpenholeUD_6101 := [[425.29, -24.3, 180.52], [-0.061977, 0.704385, 0.700279, 0.098026], [0,0,0,0], [9E9, 9E9, 9E9, 9E9, 9E9, 9E9]];
	VAR robtarget OpenholeUD_6102 := [[429.29, -24.3, 180.72], [-0.048795, 0.705421, 0.701939, 0.085337], [0,0,0,0], [9E9, 9E9, 9E9, 9E9, 9E9, 9E9]];
	VAR robtarget OpenholeUD_6103 := [[433.28, -24.3, 180.93], [-0.035432, 0.706218, 0.703389, 0.072411], [0,0,0,0], [9E9, 9E9, 9E9, 9E9, 9E9, 9E9]];
	VAR robtarget OpenholeUD_6104 := [[437.28, -24.3, 181.13], [-0.021929, 0.706767, 0.704617, 0.059284], [0,0,0,0], [9E9, 9E9, 9E9, 9E9, 9E9, 9E9]];
	VAR robtarget OpenholeUD_6105 := [[441.27, -24.3, 181.33], [-0.008327, 0.707058, 0.705609, 0.045993], [0,0,0,0], [9E9, 9E9, 9E9, 9E9, 9E9, 9E9]];
	VAR robtarget OpenholeUD_6106 := [[446.05, -24.3, 181.57], [0.008, 0.707062, 0.706472, 0.029944], [0,0,0,0], [9E9, 9E9, 9E9, 9E9, 9E9, 9E9]];
	VAR robtarget OpenholeUD_6107 := [[446.05, -24.3, 181.57], [0.008, 0.707062, 0.706472, 0.029944], [0,0,0,0], [9E9, 9E9, 9E9, 9E9, 9E9, 9E9]];
	VAR robtarget OpenholeUD_6108 := [[444.56, -23.1, 181.55], [-0.001167, 0.707106, 0.706431, 0.0309], [0,0,0,0], [9E9, 9E9, 9E9, 9E9, 9E9, 9E9]];
	VAR robtarget OpenholeUD_6109 := [[440.57, -23.1, 181.4], [-0.014813, 0.706952, 0.705717, 0.044318], [0,0,0,0], [9E9, 9E9, 9E9, 9E9, 9E9, 9E9]];
	VAR robtarget OpenholeUD_6110 := [[436.57, -23.1, 181.24], [-0.02839, 0.706537, 0.704756, 0.057611], [0,0,0,0], [9E9, 9E9, 9E9, 9E9, 9E9, 9E9]];
	VAR robtarget OpenholeUD_6111 := [[432.57, -23.1, 181.08], [-0.041854, 0.705867, 0.703559, 0.07074], [0,0,0,0], [9E9, 9E9, 9E9, 9E9, 9E9, 9E9]];
	VAR robtarget OpenholeUD_6112 := [[428.57, -23.1, 180.93], [-0.055163, 0.704952, 0.702139, 0.083667], [0,0,0,0], [9E9, 9E9, 9E9, 9E9, 9E9, 9E9]];
	VAR robtarget OpenholeUD_6113 := [[424.58, -23.1, 180.77], [-0.068278, 0.703803, 0.700511, 0.096358], [0,0,0,0], [9E9, 9E9, 9E9, 9E9, 9E9, 9E9]];
	VAR robtarget OpenholeUD_6114 := [[420.58, -23.1, 180.61], [-0.081162, 0.702433, 0.698689, 0.108784], [0,0,0,0], [9E9, 9E9, 9E9, 9E9, 9E9, 9E9]];
	VAR robtarget OpenholeUD_6115 := [[416.58, -23.1, 180.46], [-0.093785, 0.70086, 0.696692, 0.120917], [0,0,0,0], [9E9, 9E9, 9E9, 9E9, 9E9, 9E9]];
	VAR robtarget OpenholeUD_6116 := [[412.59, -23.1, 180.3], [-0.106119, 0.699099, 0.694537, 0.132736], [0,0,0,0], [9E9, 9E9, 9E9, 9E9, 9E9, 9E9]];
	VAR robtarget OpenholeUD_6117 := [[408.59, -23.1, 180.14], [-0.118141, 0.697168, 0.692243, 0.144223], [0,0,0,0], [9E9, 9E9, 9E9, 9E9, 9E9, 9E9]];
	VAR robtarget OpenholeUD_6118 := [[404.59, -23.1, 179.99], [-0.129831, 0.695085, 0.689828, 0.155363], [0,0,0,0], [9E9, 9E9, 9E9, 9E9, 9E9, 9E9]];
	VAR robtarget OpenholeUD_6119 := [[400.6, -23.1, 179.83], [-0.141176, 0.69287, 0.68731, 0.166148], [0,0,0,0], [9E9, 9E9, 9E9, 9E9, 9E9, 9E9]];
	VAR robtarget OpenholeUD_6120 := [[396.6, -23.1, 179.67], [-0.152164, 0.69054, 0.684706, 0.176571], [0,0,0,0], [9E9, 9E9, 9E9, 9E9, 9E9, 9E9]];
	VAR robtarget OpenholeUD_6121 := [[389.34, -23.1, 179.39], [-0.171188, 0.686072, 0.679812, 0.194564], [0,0,0,0], [9E9, 9E9, 9E9, 9E9, 9E9, 9E9]];
	VAR robtarget OpenholeUD_6122 := [[385.34, -23.1, 179.4], [-0.183051, 0.683002, 0.683002, 0.183051], [0,0,0,0], [9E9, 9E9, 9E9, 9E9, 9E9, 9E9]];
	VAR robtarget OpenholeUD_6123 := [[381.34, -23.1, 179.41], [-0.183051, 0.683002, 0.683002, 0.183051], [0,0,0,0], [9E9, 9E9, 9E9, 9E9, 9E9, 9E9]];
	VAR robtarget OpenholeUD_6124 := [[377.34, -23.1, 179.43], [-0.183051, 0.683002, 0.683002, 0.183051], [0,0,0,0], [9E9, 9E9, 9E9, 9E9, 9E9, 9E9]];
	VAR robtarget OpenholeUD_6125 := [[373.34, -23.1, 179.44], [-0.183051, 0.683002, 0.683002, 0.183051], [0,0,0,0], [9E9, 9E9, 9E9, 9E9, 9E9, 9E9]];
	VAR robtarget OpenholeUD_6126 := [[369.34, -23.1, 179.45], [-0.183051, 0.683002, 0.683002, 0.183051], [0,0,0,0], [9E9, 9E9, 9E9, 9E9, 9E9, 9E9]];
	VAR robtarget OpenholeUD_6127 := [[369.34, -23.1, 179.45], [-0.183051, 0.683002, 0.683002, 0.183051], [0,0,0,0], [9E9, 9E9, 9E9, 9E9, 9E9, 9E9]];
	VAR robtarget OpenholeUD_6128 := [[369.34, -21.9, 180.14], [-0.183051, 0.683002, 0.683002, 0.183051], [0,0,0,0], [9E9, 9E9, 9E9, 9E9, 9E9, 9E9]];
	VAR robtarget OpenholeUD_6129 := [[373.34, -21.9, 180.13], [-0.183051, 0.683002, 0.683002, 0.183051], [0,0,0,0], [9E9, 9E9, 9E9, 9E9, 9E9, 9E9]];
	VAR robtarget OpenholeUD_6130 := [[377.34, -21.9, 180.12], [-0.183051, 0.683002, 0.683002, 0.183051], [0,0,0,0], [9E9, 9E9, 9E9, 9E9, 9E9, 9E9]];
	VAR robtarget OpenholeUD_6131 := [[381.34, -21.9, 180.11], [-0.183051, 0.683002, 0.683002, 0.183051], [0,0,0,0], [9E9, 9E9, 9E9, 9E9, 9E9, 9E9]];
	VAR robtarget OpenholeUD_6132 := [[385.34, -21.9, 180.09], [-0.183051, 0.683002, 0.683002, 0.183051], [0,0,0,0], [9E9, 9E9, 9E9, 9E9, 9E9, 9E9]];
	VAR robtarget OpenholeUD_6133 := [[389.34, -21.9, 180.08], [-0.174625, 0.685205, 0.680774, 0.191172], [0,0,0,0], [9E9, 9E9, 9E9, 9E9, 9E9, 9E9]];
	VAR robtarget OpenholeUD_6134 := [[393.34, -21.9, 180.19], [-0.164366, 0.687738, 0.683458, 0.181342], [0,0,0,0], [9E9, 9E9, 9E9, 9E9, 9E9, 9E9]];
	VAR robtarget OpenholeUD_6135 := [[397.34, -21.9, 180.3], [-0.153739, 0.690192, 0.686083, 0.171146], [0,0,0,0], [9E9, 9E9, 9E9, 9E9, 9E9, 9E9]];
	VAR robtarget OpenholeUD_6136 := [[401.34, -21.9, 180.41], [-0.142746, 0.692549, 0.688631, 0.160586], [0,0,0,0], [9E9, 9E9, 9E9, 9E9, 9E9, 9E9]];
	VAR robtarget OpenholeUD_6137 := [[405.34, -21.9, 180.52], [-0.131397, 0.694791, 0.691086, 0.149666], [0,0,0,0], [9E9, 9E9, 9E9, 9E9, 9E9, 9E9]];
	VAR robtarget OpenholeUD_6138 := [[409.33, -21.9, 180.63], [-0.1197, 0.696902, 0.693431, 0.138394], [0,0,0,0], [9E9, 9E9, 9E9, 9E9, 9E9, 9E9]];
	VAR robtarget OpenholeUD_6139 := [[413.33, -21.9, 180.75], [-0.107672, 0.698861, 0.695648, 0.126782], [0,0,0,0], [9E9, 9E9, 9E9, 9E9, 9E9, 9E9]];
	VAR robtarget OpenholeUD_6140 := [[417.33, -21.9, 180.86], [-0.095331, 0.700651, 0.697718, 0.114844], [0,0,0,0], [9E9, 9E9, 9E9, 9E9, 9E9, 9E9]];
	VAR robtarget OpenholeUD_6141 := [[421.33, -21.9, 180.97], [-0.0827, 0.702254, 0.699624, 0.1026], [0,0,0,0], [9E9, 9E9, 9E9, 9E9, 9E9, 9E9]];
	VAR robtarget OpenholeUD_6142 := [[425.33, -21.9, 181.08], [-0.069808, 0.703652, 0.701346, 0.090073], [0,0,0,0], [9E9, 9E9, 9E9, 9E9, 9E9, 9E9]];
	VAR robtarget OpenholeUD_6143 := [[429.33, -21.9, 181.19], [-0.056687, 0.704831, 0.70287, 0.077291], [0,0,0,0], [9E9, 9E9, 9E9, 9E9, 9E9, 9E9]];
	VAR robtarget OpenholeUD_6144 := [[433.33, -21.9, 181.3], [-0.043371, 0.705775, 0.704179, 0.064285], [0,0,0,0], [9E9, 9E9, 9E9, 9E9, 9E9, 9E9]];
	VAR robtarget OpenholeUD_6145 := [[437.32, -21.9, 181.41], [-0.029902, 0.706474, 0.705259, 0.051091], [0,0,0,0], [9E9, 9E9, 9E9, 9E9, 9E9, 9E9]];
	VAR robtarget OpenholeUD_6146 := [[443.69, -21.9, 181.58], [-0.008244, 0.707059, 0.706479, 0.029791], [0,0,0,0], [9E9, 9E9, 9E9, 9E9, 9E9, 9E9]];
	VAR robtarget OpenholeUD_6147 := [[443.69, -21.9, 181.58], [-0.008244, 0.707059, 0.706479, 0.029791], [0,0,0,0], [9E9, 9E9, 9E9, 9E9, 9E9, 9E9]];
	VAR robtarget OpenholeUD_6148 := [[443.16, -20.7, 181.64], [-0.014137, 0.706965, 0.706571, 0.027514], [0,0,0,0], [9E9, 9E9, 9E9, 9E9, 9E9, 9E9]];
	VAR robtarget OpenholeUD_6149 := [[439.16, -20.7, 181.58], [-0.027746, 0.706562, 0.705921, 0.040934], [0,0,0,0], [9E9, 9E9, 9E9, 9E9, 9E9, 9E9]];
	VAR robtarget OpenholeUD_6150 := [[435.16, -20.7, 181.51], [-0.041255, 0.705902, 0.705024, 0.054229], [0,0,0,0], [9E9, 9E9, 9E9, 9E9, 9E9, 9E9]];
	VAR robtarget OpenholeUD_6151 := [[431.16, -20.7, 181.45], [-0.054621, 0.704994, 0.703891, 0.06736], [0,0,0,0], [9E9, 9E9, 9E9, 9E9, 9E9, 9E9]];
	VAR robtarget OpenholeUD_6152 := [[427.16, -20.7, 181.38], [-0.067805, 0.703848, 0.702534, 0.080288], [0,0,0,0], [9E9, 9E9, 9E9, 9E9, 9E9, 9E9]];
	VAR robtarget OpenholeUD_6153 := [[423.16, -20.7, 181.32], [-0.080769, 0.702479, 0.700967, 0.092981], [0,0,0,0], [9E9, 9E9, 9E9, 9E9, 9E9, 9E9]];
	VAR robtarget OpenholeUD_6154 := [[419.17, -20.7, 181.26], [-0.093479, 0.700901, 0.699206, 0.105408], [0,0,0,0], [9E9, 9E9, 9E9, 9E9, 9E9, 9E9]];
	VAR robtarget OpenholeUD_6155 := [[415.17, -20.7, 181.19], [-0.105907, 0.699131, 0.697268, 0.117544], [0,0,0,0], [9E9, 9E9, 9E9, 9E9, 9E9, 9E9]];
	VAR robtarget OpenholeUD_6156 := [[411.17, -20.7, 181.13], [-0.118028, 0.697187, 0.695172, 0.129367], [0,0,0,0], [9E9, 9E9, 9E9, 9E9, 9E9, 9E9]];
	VAR robtarget OpenholeUD_6157 := [[407.17, -20.7, 181.06], [-0.129822, 0.695087, 0.692935, 0.140859], [0,0,0,0], [9E9, 9E9, 9E9, 9E9, 9E9, 9E9]];
	VAR robtarget OpenholeUD_6158 := [[403.17, -20.7, 181], [-0.141271, 0.692851, 0.690575, 0.152007], [0,0,0,0], [9E9, 9E9, 9E9, 9E9, 9E9, 9E9]];
